LIN {X 0,Y 275.773,Z 716.506,A -85,B 0,C 180,E1 16932.937,E2 16932.937} C_VEL
LIN {X 0,Y 278.807,Z 722.231,A -85,B 0,C 180,E1 16937.514,E2 16937.514} C_VEL
LIN {X 0,Y 285.575,Z 736.206,A -85,B 0,C 180,E1 16944.998,E2 16944.998} C_VEL
LIN {X 0,Y 292.678,Z 753.38,A -85,B 0,C 180,E1 16951.647,E2 16951.647} C_VEL
LIN {X 0,Y 298.576,Z 772.807,A -85,B 0,C 180,E1 16957.666,E2 16957.666} C_VEL
LIN {X 0,Y 301.91,Z 794.325,A -85,B 0,C 180,E1 16963.416,E2 16963.416} C_VEL
LIN {X 0,Y 302.06,Z 807.18,A -85,B 0,C 180,E1 16966.628,E2 16966.628} C_VEL
LIN {X 0,Y 289.061,Z 835.016,A -85,B 0,C 180,E1 16971.838,E2 16971.838} C_VEL
LIN {X 0,Y 277.029,Z 857.298,A -85,B 0,C 180,E1 16977.972,E2 16977.972} C_VEL
LIN {X 0,Y 266.798,Z 875.138,A -85,B 0,C 180,E1 16985.37,E2 16985.37} C_VEL
LIN {X 0,Y 260.131,Z 886.98,A -85,B 0,C 180,E1 16993.139,E2 16993.139} C_VEL
LIN {X 0,Y 257.066,Z 893.034,A -85,B 0,C 180,E1 16999.857,E2 16999.857} C_VEL
LIN {X 0,Y 255.939,Z 895.924,A -85,B 0,C 180,E1 17006.62,E2 17006.62} C_VEL
LIN {X 0,Y 255.938,Z 895.892,A -85,B 0,C 180,E1 17013.38,E2 17013.38} C_VEL
LIN {X 0,Y 257.68,Z 891.722,A -85,B 0,C 180,E1 17021.827,E2 17021.827} C_VEL
LIN {X 0,Y 262.63,Z 882.447,A -85,B 0,C 180,E1 17030.166,E2 17030.166} C_VEL
LIN {X 0,Y 271.349,Z 867.242,A -85,B 0,C 180,E1 17038.209,E2 17038.209} C_VEL
LIN {X 0,Y 282.59,Z 847.082,A -85,B 0,C 180,E1 17045.032,E2 17045.032} C_VEL
LIN {X 0,Y 294.293,Z 824.104,A -85,B 0,C 180,E1 17050.34,E2 17050.34} C_VEL
LIN {X 0,Y 302.608,Z 805.568,A -85,B 0,C 180,E1 17053.512,E2 17053.512} C_VEL
LIN {X 0,Y 300.613,Z 783.565,A -85,B 0,C 180,E1 17059.276,E2 17059.276} C_VEL
LIN {X 0,Y 295.972,Z 763.231,A -85,B 0,C 180,E1 17065.01,E2 17065.01} C_VEL
LIN {X 0,Y 289.142,Z 744.349,A -85,B 0,C 180,E1 17071.442,E2 17071.442} C_VEL
LIN {X 0,Y 281.784,Z 728.351,A -85,B 0,C 180,E1 17078.651,E2 17078.651} C_VEL
LIN {X 0,Y 278.046,Z 721.516,A -85,B 0,C 180,E1 17083.047,E2 17083.047} C_VEL
LIN {X 0,Y 275.21,Z 715.444,A -85,B 0,C 180,E1 17087.74,E2 17087.74} C_VEL
LIN {X 0,Y 272.952,Z 711.906,A -85,B 0,C 180,E1 17098.422,E2 17098.422} C_VEL
LIN {X 0,Y 276.968,Z 716.793,A -85,B 0,C 180,E1 17107.559,E2 17107.559} C_VEL
LIN {X 0,Y 281.856,Z 725.008,A -85,B 0,C 180,E1 17113.023,E2 17113.023} C_VEL
LIN {X 0,Y 289.079,Z 736.426,A -85,B 0,C 180,E1 17118.645,E2 17118.645} C_VEL
LIN {X 0,Y 298.908,Z 754.882,A -85,B 0,C 180,E1 17124.806,E2 17124.806} C_VEL
LIN {X 0,Y 308.931,Z 777.729,A -85,B 0,C 180,E1 17130.453,E2 17130.453} C_VEL
LIN {X 0,Y 316.347,Z 802.298,A -85,B 0,C 180,E1 17135.213,E2 17135.213} C_VEL
LIN {X 0,Y 304.344,Z 840.414,A -85,B 0,C 180,E1 17138.476,E2 17138.476} C_VEL
LIN {X 0,Y 290.625,Z 875.361,A -85,B 0,C 180,E1 17142.899,E2 17142.899} C_VEL
LIN {X 0,Y 278.063,Z 904.903,A -85,B 0,C 180,E1 17148.334,E2 17148.334} C_VEL
LIN {X 0,Y 267.214,Z 930.489,A -85,B 0,C 180,E1 17154.988,E2 17154.988} C_VEL
LIN {X 0,Y 259.237,Z 951.979,A -85,B 0,C 180,E1 17162.904,E2 17162.904} C_VEL
LIN {X 0,Y 255.098,Z 967.514,A -85,B 0,C 180,E1 17171.173,E2 17171.173} C_VEL
LIN {X 0,Y 254.243,Z 975.961,A -85,B 0,C 180,E1 17177.835,E2 17177.835} C_VEL
LIN {X 0,Y 254.275,Z 980.166,A -85,B 0,C 180,E1 17183.183,E2 17183.183} C_VEL
LIN {X 0,Y 254.787,Z 982.267,A -85,B 0,C 180,E1 17190,E2 17190} C_VEL
LIN {X 0,Y 254.269,Z 980.175,A -85,B 0,C 180,E1 17196.817,E2 17196.817} C_VEL
LIN {X 0,Y 254.36,Z 973.333,A -85,B 0,C 180,E1 17204.604,E2 17204.604} C_VEL
LIN {X 0,Y 256.876,Z 959.841,A -85,B 0,C 180,E1 17213.361,E2 17213.361} C_VEL
LIN {X 0,Y 263.615,Z 939.724,A -85,B 0,C 180,E1 17221.971,E2 17221.971} C_VEL
LIN {X 0,Y 273.628,Z 915.458,A -85,B 0,C 180,E1 17229.203,E2 17229.203} C_VEL
LIN {X 0,Y 285.643,Z 887.471,A -85,B 0,C 180,E1 17235.11,E2 17235.11} C_VEL
LIN {X 0,Y 298.673,Z 855.592,A -85,B 0,C 180,E1 17239.823,E2 17239.823} C_VEL
LIN {X 0,Y 311.279,Z 820.186,A -85,B 0,C 180,E1 17243.408,E2 17243.408} C_VEL
LIN {X 0,Y 316.34,Z 802.002,A -85,B 0,C 180,E1 17244.859,E2 17244.859} C_VEL
LIN {X 0,Y 308.472,Z 776.099,A -85,B 0,C 180,E1 17249.903,E2 17249.903} C_VEL
LIN {X 0,Y 298.548,Z 753.828,A -85,B 0,C 180,E1 17255.505,E2 17255.505} C_VEL
LIN {X 0,Y 289.965,Z 738.122,A -85,B 0,C 180,E1 17260.822,E2 17260.822} C_VEL
LIN {X 0,Y 286.089,Z 736.306,A -85,B 0,C 180,E1 17262.977,E2 17262.977} C_VEL
LIN {X 0,Y 282.076,Z 736.045,A -85,B 0,C 180,E1 17265.282,E2 17265.282} C_VEL
LIN {X 0,Y 277.56,Z 729.06,A -85,B 0,C 180,E1 17269.674,E2 17269.674} C_VEL
LIN {X 0,Y 274.527,Z 723.198,A -85,B 0,C 180,E1 17274.079,E2 17274.079} C_VEL
LIN {X 0,Y 271.676,Z 719.971,A -85,B 0,C 180,E1 17281.181,E2 17281.181} C_VEL
LIN {X 0,Y 273.643,Z 723.735,A -85,B 0,C 180,E1 17292.432,E2 17292.432} C_VEL
LIN {X 0,Y 276.931,Z 731.578,A -85,B 0,C 180,E1 17298.252,E2 17298.252} C_VEL
LIN {X 0,Y 282.749,Z 744.678,A -85,B 0,C 180,E1 17305.266,E2 17305.266} C_VEL
LIN {X 0,Y 289.066,Z 761.562,A -85,B 0,C 180,E1 17311.901,E2 17311.901} C_VEL
LIN {X 0,Y 293.94,Z 781.055,A -85,B 0,C 180,E1 17318.017,E2 17318.017} C_VEL
LIN {X 0,Y 296.249,Z 803.118,A -85,B 0,C 180,E1 17324.083,E2 17324.083} C_VEL
LIN {X 0,Y 296.074,Z 809.506,A -85,B 0,C 180,E1 17325.739,E2 17325.739} C_VEL
LIN {X 0,Y 282.768,Z 836.72,A -85,B 0,C 180,E1 17330.943,E2 17330.943} C_VEL
LIN {X 0,Y 270.767,Z 858.109,A -85,B 0,C 180,E1 17336.916,E2 17336.916} C_VEL
LIN {X 0,Y 260.508,Z 875.122,A -85,B 0,C 180,E1 17343.949,E2 17343.949} C_VEL
LIN {X 0,Y 253.25,Z 887.277,A -85,B 0,C 180,E1 17351.771,E2 17351.771} C_VEL
LIN {X 0,Y 249.383,Z 894.348,A -85,B 0,C 180,E1 17359.541,E2 17359.541} C_VEL
LIN {X 0,Y 248.179,Z 897.233,A -85,B 0,C 180,E1 17366.514,E2 17366.514} C_VEL
LIN {X 0,Y 248.178,Z 897.201,A -85,B 0,C 180,E1 17373.486,E2 17373.486} C_VEL
LIN {X 0,Y 250.034,Z 893.041,A -85,B 0,C 180,E1 17382.194,E2 17382.194} C_VEL
LIN {X 0,Y 255.287,Z 883.772,A -85,B 0,C 180,E1 17390.772,E2 17390.772} C_VEL
LIN {X 0,Y 264.48,Z 868.573,A -85,B 0,C 180,E1 17399.01,E2 17399.01} C_VEL
LIN {X 0,Y 276.236,Z 848.436,A -85,B 0,C 180,E1 17405.961,E2 17405.961} C_VEL
LIN {X 0,Y 289.303,Z 823.666,A -85,B 0,C 180,E1 17411.685,E2 17411.685} C_VEL
LIN {X 0,Y 296.309,Z 807.713,A -85,B 0,C 180,E1 17414.535,E2 17414.535} C_VEL
LIN {X 0,Y 294.553,Z 785.102,A -85,B 0,C 180,E1 17420.725,E2 17420.725} C_VEL
LIN {X 0,Y 289.975,Z 764.717,A -85,B 0,C 180,E1 17426.887,E2 17426.887} C_VEL
LIN {X 0,Y 283.421,Z 746.135,A -85,B 0,C 180,E1 17433.851,E2 17433.851} C_VEL
LIN {X 0,Y 278.14,Z 734.597,A -85,B 0,C 180,E1 17439.737,E2 17439.737} C_VEL
LIN {X 0,Y 275.601,Z 728.908,A -85,B 0,C 180,E1 17443.302,E2 17443.302} C_VEL
LIN {X 0,Y 273.167,Z 723.013,A -85,B 0,C 180,E1 17448.052,E2 17448.052} C_VEL
LIN {X 0,Y 271.215,Z 719.663,A -85,B 0,C 180,E1 17456.817,E2 17456.817} C_VEL
LIN {X 0,Y 272.921,Z 722.001,A -85,B 0,C 180,E1 17463.622,E2 17463.622} C_VEL
LIN {X 0,Y 275.18,Z 724.57,A -85,B 0,C 180,E1 17467.311,E2 17467.311} C_VEL
LIN {X 0,Y 279.588,Z 732.408,A -85,B 0,C 180,E1 17472.652,E2 17472.652} C_VEL
LIN {X 0,Y 286.344,Z 743.669,A -85,B 0,C 180,E1 17478.239,E2 17478.239} C_VEL
LIN {X 0,Y 295.044,Z 760.875,A -85,B 0,C 180,E1 17484.156,E2 17484.156} C_VEL
LIN {X 0,Y 304.381,Z 783.881,A -85,B 0,C 180,E1 17490.025,E2 17490.025} C_VEL
LIN {X 0,Y 310.331,Z 804.847,A -85,B 0,C 180,E1 17494.246,E2 17494.246} C_VEL
LIN {X 0,Y 298.164,Z 841.829,A -85,B 0,C 180,E1 17497.569,E2 17497.569} C_VEL
LIN {X 0,Y 284.226,Z 875.806,A -85,B 0,C 180,E1 17501.989,E2 17501.989} C_VEL
LIN {X 0,Y 271.005,Z 905.4,A -85,B 0,C 180,E1 17507.607,E2 17507.607} C_VEL
LIN {X 0,Y 259.166,Z 932.085,A -85,B 0,C 180,E1 17514.902,E2 17514.902} C_VEL
LIN {X 0,Y 251.03,Z 953.123,A -85,B 0,C 180,E1 17523.202,E2 17523.202} C_VEL
LIN {X 0,Y 246.974,Z 968.527,A -85,B 0,C 180,E1 17532.212,E2 17532.212} C_VEL
LIN {X 0,Y 246.378,Z 976.356,A -85,B 0,C 180,E1 17539.412,E2 17539.412} C_VEL
LIN {X 0,Y 246.673,Z 980.374,A -85,B 0,C 180,E1 17546.493,E2 17546.493} C_VEL
LIN {X 0,Y 246.995,Z 980.955,A -85,B 0,C 180,E1 17550,E2 17550} C_VEL
LIN {X 0,Y 246.432,Z 978.846,A -85,B 0,C 180,E1 17557.035,E2 17557.035} C_VEL
LIN {X 0,Y 246.568,Z 971.973,A -85,B 0,C 180,E1 17565.076,E2 17565.076} C_VEL
LIN {X 0,Y 249.374,Z 958.451,A -85,B 0,C 180,E1 17574.107,E2 17574.107} C_VEL
LIN {X 0,Y 256.602,Z 938.302,A -85,B 0,C 180,E1 17582.954,E2 17582.954} C_VEL
LIN {X 0,Y 266.993,Z 914.605,A -85,B 0,C 180,E1 17590.179,E2 17590.179} C_VEL
LIN {X 0,Y 280.023,Z 885.552,A -85,B 0,C 180,E1 17596.396,E2 17596.396} C_VEL
LIN {X 0,Y 293.699,Z 853.458,A -85,B 0,C 180,E1 17601.123,E2 17601.123} C_VEL
LIN {X 0,Y 307.066,Z 816.863,A -85,B 0,C 180,E1 17604.776,E2 17604.776} C_VEL
LIN {X 0,Y 310.458,Z 805.145,A -85,B 0,C 180,E1 17605.719,E2 17605.719} C_VEL
LIN {X 0,Y 303.059,Z 779.517,A -85,B 0,C 180,E1 17610.953,E2 17610.953} C_VEL
LIN {X 0,Y 293.585,Z 757.473,A -85,B 0,C 180,E1 17616.879,E2 17616.879} C_VEL
LIN {X 0,Y 284.72,Z 740.905,A -85,B 0,C 180,E1 17623.072,E2 17623.072} C_VEL
LIN {X 0,Y 282.076,Z 736.045,A -85,B 0,C 180,E1 17625.282,E2 17625.282} C_VEL
LIN {X 0,Y 273.842,Z 734.194,A -85,B 0,C 180,E1 17631.882,E2 17631.882} C_VEL
LIN {X 0,Y 273.556,Z 733.6,A -85,B 0,C 180,E1 17632.32,E2 17632.32} C_VEL
LIN {X 0,Y 272.416,Z 730.73,A -85,B 0,C 180,E1 17634.431,E2 17634.431} C_VEL
LIN {X 0,Y 269.829,Z 727.655,A -85,B 0,C 180,E1 17641.189,E2 17641.189} C_VEL
LIN {X 0,Y 271.298,Z 731.406,A -85,B 0,C 180,E1 17652.236,E2 17652.236} C_VEL
LIN {X 0,Y 276.241,Z 743.627,A -85,B 0,C 180,E1 17660.957,E2 17660.957} C_VEL
LIN {X 0,Y 282.102,Z 759.424,A -85,B 0,C 180,E1 17668.333,E2 17668.333} C_VEL
LIN {X 0,Y 287.086,Z 777.8,A -85,B 0,C 180,E1 17674.862,E2 17674.862} C_VEL
LIN {X 0,Y 289.601,Z 795.656,A -85,B 0,C 180,E1 17680.221,E2 17680.221} C_VEL
LIN {X 0,Y 289.774,Z 812.608,A -85,B 0,C 180,E1 17684.944,E2 17684.944} C_VEL
LIN {X 0,Y 276.676,Z 838.218,A -85,B 0,C 180,E1 17689.961,E2 17689.961} C_VEL
LIN {X 0,Y 264.236,Z 859.448,A -85,B 0,C 180,E1 17695.988,E2 17695.988} C_VEL
LIN {X 0,Y 252.723,Z 877.646,A -85,B 0,C 180,E1 17703.809,E2 17703.809} C_VEL
LIN {X 0,Y 245.203,Z 889.619,A -85,B 0,C 180,E1 17712.079,E2 17712.079} C_VEL
LIN {X 0,Y 241.706,Z 895.663,A -85,B 0,C 180,E1 17719.205,E2 17719.205} C_VEL
LIN {X 0,Y 240.404,Z 898.544,A -85,B 0,C 180,E1 17726.401,E2 17726.401} C_VEL
LIN {X 0,Y 240.404,Z 898.513,A -85,B 0,C 180,E1 17733.599,E2 17733.599} C_VEL
LIN {X 0,Y 242.405,Z 894.357,A -85,B 0,C 180,E1 17742.584,E2 17742.584} C_VEL
LIN {X 0,Y 247.994,Z 885.093,A -85,B 0,C 180,E1 17751.413,E2 17751.413} C_VEL
LIN {X 0,Y 257.672,Z 869.902,A -85,B 0,C 180,E1 17759.853,E2 17759.853} C_VEL
LIN {X 0,Y 269.956,Z 849.787,A -85,B 0,C 180,E1 17766.934,E2 17766.934} C_VEL
LIN {X 0,Y 283.533,Z 825.049,A -85,B 0,C 180,E1 17772.732,E2 17772.732} C_VEL
LIN {X 0,Y 290.1,Z 810.596,A -85,B 0,C 180,E1 17775.402,E2 17775.402} C_VEL
LIN {X 0,Y 288.869,Z 788.876,A -85,B 0,C 180,E1 17781.589,E2 17781.589} C_VEL
LIN {X 0,Y 285.281,Z 770.474,A -85,B 0,C 180,E1 17787.424,E2 17787.424} C_VEL
LIN {X 0,Y 279.61,Z 752.493,A -85,B 0,C 180,E1 17794.43,E2 17794.43} C_VEL
LIN {X 0,Y 274.685,Z 740.648,A -85,B 0,C 180,E1 17800.763,E2 17800.763} C_VEL
LIN {X 0,Y 272.75,Z 735.962,A -85,B 0,C 180,E1 17803.949,E2 17803.949} C_VEL
LIN {X 0,Y 270.656,Z 730.403,A -85,B 0,C 180,E1 17808.754,E2 17808.754} C_VEL
LIN {X 0,Y 269.534,Z 727.451,A -85,B 0,C 180,E1 17818.402,E2 17818.402} C_VEL
LIN {X 0,Y 272.989,Z 731.942,A -85,B 0,C 180,E1 17826.891,E2 17826.891} C_VEL
LIN {X 0,Y 277.382,Z 740.093,A -85,B 0,C 180,E1 17832.474,E2 17832.474} C_VEL
LIN {X 0,Y 283.65,Z 751.509,A -85,B 0,C 180,E1 17838.117,E2 17838.117} C_VEL
LIN {X 0,Y 292.288,Z 769.765,A -85,B 0,C 180,E1 17844.399,E2 17844.399} C_VEL
LIN {X 0,Y 299.943,Z 790.603,A -85,B 0,C 180,E1 17849.727,E2 17849.727} C_VEL
LIN {X 0,Y 304.516,Z 808.446,A -85,B 0,C 180,E1 17853.46,E2 17853.46} C_VEL
LIN {X 0,Y 291.73,Z 844.092,A -85,B 0,C 180,E1 17856.717,E2 17856.717} C_VEL
LIN {X 0,Y 277.252,Z 877.65,A -85,B 0,C 180,E1 17861.256,E2 17861.256} C_VEL
LIN {X 0,Y 262.431,Z 909.204,A -85,B 0,C 180,E1 17867.636,E2 17867.636} C_VEL
LIN {X 0,Y 250.611,Z 934.587,A -85,B 0,C 180,E1 17875.189,E2 17875.189} C_VEL
LIN {X 0,Y 242.975,Z 953.491,A -85,B 0,C 180,E1 17883.24,E2 17883.24} C_VEL
LIN {X 0,Y 239.025,Z 968.3,A -85,B 0,C 180,E1 17892.55,E2 17892.55} C_VEL
LIN {X 0,Y 238.545,Z 976.432,A -85,B 0,C 180,E1 17900.901,E2 17900.901} C_VEL
LIN {X 0,Y 238.866,Z 979.056,A -85,B 0,C 180,E1 17906.378,E2 17906.378} C_VEL
LIN {X 0,Y 239.194,Z 979.642,A -85,B 0,C 180,E1 17910,E2 17910} C_VEL
LIN {X 0,Y 238.593,Z 977.515,A -85,B 0,C 180,E1 17917.267,E2 17917.267} C_VEL
LIN {X 0,Y 238.805,Z 970.615,A -85,B 0,C 180,E1 17925.578,E2 17925.578} C_VEL
LIN {X 0,Y 241.829,Z 957.133,A -85,B 0,C 180,E1 17934.862,E2 17934.862} C_VEL
LIN {X 0,Y 249.599,Z 936.935,A -85,B 0,C 180,E1 17943.976,E2 17943.976} C_VEL
LIN {X 0,Y 260.742,Z 913.024,A -85,B 0,C 180,E1 17951.395,E2 17951.395} C_VEL
LIN {X 0,Y 273.892,Z 885.103,A -85,B 0,C 180,E1 17957.467,E2 17957.467} C_VEL
LIN {X 0,Y 288.069,Z 853.225,A -85,B 0,C 180,E1 17962.234,E2 17962.234} C_VEL
LIN {X 0,Y 301.44,Z 818.115,A -85,B 0,C 180,E1 17965.798,E2 17965.798} C_VEL
LIN {X 0,Y 304.447,Z 807.665,A -85,B 0,C 180,E1 17966.71,E2 17966.71} C_VEL
LIN {X 0,Y 297.663,Z 783.084,A -85,B 0,C 180,E1 17972.031,E2 17972.031} C_VEL
LIN {X 0,Y 289.298,Z 762.856,A -85,B 0,C 180,E1 17977.776,E2 17977.776} C_VEL
LIN {X 0,Y 281.617,Z 747.621,A -85,B 0,C 180,E1 17983.669,E2 17983.669} C_VEL
LIN {X 0,Y 275.493,Z 736.621,A -85,B 0,C 180,E1 17989.831,E2 17989.831} C_VEL
LIN {X 0,Y 273.556,Z 733.6,A -85,B 0,C 180,E1 17992.32,E2 17992.32} C_VEL
LIN {X 0,Y 271.902,Z 733.916,A -85,B 0,C 180,E1 17994.118,E2 17994.118} C_VEL
LIN {X 0,Y 269.049,Z 737.187,A -85,B 0,C 180,E1 17996.855,E2 17996.855} C_VEL
LIN {X 0,Y 268.887,Z 737.1,A -85,B 0,C 180,E1 17997.174,E2 17997.174} C_VEL
LIN {X 0,Y 267.483,Z 735.272,A -85,B 0,C 180,E1 18003.228,E2 18003.228} C_VEL
LIN {X 0,Y 268.824,Z 739.224,A -85,B 0,C 180,E1 18012.144,E2 18012.144} C_VEL
LIN {X 0,Y 272.607,Z 749.793,A -85,B 0,C 180,E1 18020.096,E2 18020.096} C_VEL
LIN {X 0,Y 277.39,Z 764.046,A -85,B 0,C 180,E1 18027.168,E2 18027.168} C_VEL
LIN {X 0,Y 281.67,Z 781.506,A -85,B 0,C 180,E1 18033.757,E2 18033.757} C_VEL
LIN {X 0,Y 283.808,Z 800.155,A -85,B 0,C 180,E1 18039.634,E2 18039.634} C_VEL
LIN {X 0,Y 283.745,Z 815.144,A -85,B 0,C 180,E1 18044.028,E2 18044.028} C_VEL
LIN {X 0,Y 270.039,Z 840.765,A -85,B 0,C 180,E1 18049.189,E2 18049.189} C_VEL
LIN {X 0,Y 256.886,Z 862.177,A -85,B 0,C 180,E1 18055.518,E2 18055.518} C_VEL
LIN {X 0,Y 245.244,Z 879.716,A -85,B 0,C 180,E1 18063.413,E2 18063.413} C_VEL
LIN {X 0,Y 236.918,Z 892.249,A -85,B 0,C 180,E1 18072.784,E2 18072.784} C_VEL
LIN {X 0,Y 233.073,Z 898.782,A -85,B 0,C 180,E1 18082.56,E2 18082.56} C_VEL
LIN {X 0,Y 232.297,Z 900.265,A -85,B 0,C 180,E1 18090,E2 18090} C_VEL
LIN {X 0,Y 233.075,Z 898.729,A -85,B 0,C 180,E1 18097.44,E2 18097.44} C_VEL
LIN {X 0,Y 237.02,Z 892.057,A -85,B 0,C 180,E1 18107.295,E2 18107.295} C_VEL
LIN {X 0,Y 245.408,Z 879.388,A -85,B 0,C 180,E1 18116.639,E2 18116.639} C_VEL
LIN {X 0,Y 257.207,Z 861.555,A -85,B 0,C 180,E1 18124.586,E2 18124.586} C_VEL
LIN {X 0,Y 270.968,Z 838.952,A -85,B 0,C 180,E1 18131.15,E2 18131.15} C_VEL
LIN {X 0,Y 283.915,Z 814.155,A -85,B 0,C 180,E1 18136.091,E2 18136.091} C_VEL
LIN {X 0,Y 283.262,Z 792.822,A -85,B 0,C 180,E1 18142.432,E2 18142.432} C_VEL
LIN {X 0,Y 279.983,Z 773.942,A -85,B 0,C 180,E1 18148.762,E2 18148.762} C_VEL
LIN {X 0,Y 275.729,Z 758.969,A -85,B 0,C 180,E1 18154.913,E2 18154.913} C_VEL
LIN {X 0,Y 270.832,Z 744.586,A -85,B 0,C 180,E1 18162.916,E2 18162.916} C_VEL
LIN {X 0,Y 268.459,Z 737.983,A -85,B 0,C 180,E1 18168.661,E2 18168.661} C_VEL
LIN {X 0,Y 267.498,Z 735.067,A -85,B 0,C 180,E1 18178.39,E2 18178.39} C_VEL
LIN {X 0,Y 270.718,Z 739.485,A -85,B 0,C 180,E1 18186.607,E2 18186.607} C_VEL
LIN {X 0,Y 274.933,Z 747.802,A -85,B 0,C 180,E1 18192.385,E2 18192.385} C_VEL
LIN {X 0,Y 281.753,Z 760.881,A -85,B 0,C 180,E1 18198.749,E2 18198.749} C_VEL
LIN {X 0,Y 289.78,Z 780.082,A -85,B 0,C 180,E1 18205.077,E2 18205.077} C_VEL
LIN {X 0,Y 296.653,Z 802.266,A -85,B 0,C 180,E1 18210.579,E2 18210.579} C_VEL
LIN {X 0,Y 298.485,Z 811.961,A -85,B 0,C 180,E1 18212.564,E2 18212.564} C_VEL
LIN {X 0,Y 284.132,Z 849.211,A -85,B 0,C 180,E1 18216.165,E2 18216.165} C_VEL
LIN {X 0,Y 268.819,Z 882.478,A -85,B 0,C 180,E1 18221.036,E2 18221.036} C_VEL
LIN {X 0,Y 254.307,Z 911.835,A -85,B 0,C 180,E1 18227.444,E2 18227.444} C_VEL
LIN {X 0,Y 242.454,Z 936.101,A -85,B 0,C 180,E1 18235.17,E2 18235.17} C_VEL
LIN {X 0,Y 234.193,Z 955.97,A -85,B 0,C 180,E1 18244.439,E2 18244.439} C_VEL
LIN {X 0,Y 230.969,Z 969.219,A -85,B 0,C 180,E1 18253.879,E2 18253.879} C_VEL
LIN {X 0,Y 230.764,Z 976.174,A -85,B 0,C 180,E1 18262.485,E2 18262.485} C_VEL
LIN {X 0,Y 231.4,Z 978.33,A -85,B 0,C 180,E1 18270,E2 18270} C_VEL
LIN {X 0,Y 230.754,Z 976.184,A -85,B 0,C 180,E1 18277.515,E2 18277.515} C_VEL
LIN {X 0,Y 231.002,Z 969.247,A -85,B 0,C 180,E1 18286.119,E2 18286.119} C_VEL
LIN {X 0,Y 234.545,Z 955.112,A -85,B 0,C 180,E1 18296.05,E2 18296.05} C_VEL
LIN {X 0,Y 242.414,Z 936.109,A -85,B 0,C 180,E1 18304.854,E2 18304.854} C_VEL
LIN {X 0,Y 254.876,Z 910.809,A -85,B 0,C 180,E1 18312.845,E2 18312.845} C_VEL
LIN {X 0,Y 268.914,Z 882.626,A -85,B 0,C 180,E1 18318.941,E2 18318.941} C_VEL
LIN {X 0,Y 283.532,Z 850.753,A -85,B 0,C 180,E1 18323.667,E2 18323.667} C_VEL
LIN {X 0,Y 297.869,Z 814.005,A -85,B 0,C 180,E1 18327.3,E2 18327.3} C_VEL
LIN {X 0,Y 298.219,Z 808.718,A -85,B 0,C 180,E1 18328.043,E2 18328.043} C_VEL
LIN {X 0,Y 291.884,Z 785.192,A -85,B 0,C 180,E1 18333.519,E2 18333.519} C_VEL
LIN {X 0,Y 283.675,Z 765.047,A -85,B 0,C 180,E1 18339.767,E2 18339.767} C_VEL
LIN {X 0,Y 276.216,Z 749.889,A -85,B 0,C 180,E1 18346.469,E2 18346.469} C_VEL
LIN {X 0,Y 272.499,Z 743.381,A -85,B 0,C 180,E1 18350.733,E2 18350.733} C_VEL
LIN {X 0,Y 270.161,Z 738.234,A -85,B 0,C 180,E1 18354.787,E2 18354.787} C_VEL
LIN {X 0,Y 268.887,Z 737.1,A -85,B 0,C 180,E1 18357.174,E2 18357.174} C_VEL
LIN {X 0,Y 267.305,Z 738.248,A -85,B 0,C 180,E1 18359.937,E2 18359.937} C_VEL
LIN {X 0,Y 265.042,Z 743.301,A -85,B 0,C 180,E1 18364.565,E2 18364.565} C_VEL
LIN {X 0,Y 266.082,Z 745.892,A -85,B 0,C 180,E1 18371.335,E2 18371.335} C_VEL
LIN {X 0,Y 269.217,Z 756.616,A -85,B 0,C 180,E1 18379.644,E2 18379.644} C_VEL
LIN {X 0,Y 273.203,Z 770.441,A -85,B 0,C 180,E1 18386.745,E2 18386.745} C_VEL
LIN {X 0,Y 276.695,Z 787.513,A -85,B 0,C 180,E1 18393.415,E2 18393.415} C_VEL
LIN {X 0,Y 278.058,Z 804.942,A -85,B 0,C 180,E1 18399.113,E2 18399.113} C_VEL
LIN {X 0,Y 277.595,Z 818.011,A -85,B 0,C 180,E1 18403.121,E2 18403.121} C_VEL
LIN {X 0,Y 263.019,Z 844.041,A -85,B 0,C 180,E1 18408.562,E2 18408.562} C_VEL
LIN {X 0,Y 248.596,Z 866.341,A -85,B 0,C 180,E1 18415.552,E2 18415.552} C_VEL
LIN {X 0,Y 237.16,Z 882.652,A -85,B 0,C 180,E1 18423.552,E2 18423.552} C_VEL
LIN {X 0,Y 229.46,Z 893.567,A -85,B 0,C 180,E1 18432.206,E2 18432.206} C_VEL
LIN {X 0,Y 225.329,Z 900.097,A -85,B 0,C 180,E1 18442.303,E2 18442.303} C_VEL
LIN {X 0,Y 224.537,Z 901.572,A -85,B 0,C 180,E1 18450,E2 18450} C_VEL
LIN {X 0,Y 225.333,Z 900.045,A -85,B 0,C 180,E1 18457.697,E2 18457.697} C_VEL
LIN {X 0,Y 229.569,Z 893.374,A -85,B 0,C 180,E1 18467.875,E2 18467.875} C_VEL
LIN {X 0,Y 238.192,Z 881.066,A -85,B 0,C 180,E1 18477.289,E2 18477.289} C_VEL
LIN {X 0,Y 249.824,Z 864.392,A -85,B 0,C 180,E1 18485.045,E2 18485.045} C_VEL
LIN {X 0,Y 263.223,Z 843.437,A -85,B 0,C 180,E1 18491.488,E2 18491.488} C_VEL
LIN {X 0,Y 277.695,Z 817.608,A -85,B 0,C 180,E1 18496.831,E2 18496.831} C_VEL
LIN {X 0,Y 277.819,Z 798.36,A -85,B 0,C 180,E1 18502.813,E2 18502.813} C_VEL
LIN {X 0,Y 275.261,Z 779.684,A -85,B 0,C 180,E1 18509.314,E2 18509.314} C_VEL
LIN {X 0,Y 271.483,Z 764.455,A -85,B 0,C 180,E1 18515.896,E2 18515.896} C_VEL
LIN {X 0,Y 267.509,Z 751.28,A -85,B 0,C 180,E1 18523.625,E2 18523.625} C_VEL
LIN {X 0,Y 265.849,Z 745.557,A -85,B 0,C 180,E1 18528.743,E2 18528.743} C_VEL
LIN {X 0,Y 265.074,Z 742.573,A -85,B 0,C 180,E1 18536.743,E2 18536.743} C_VEL
LIN {X 0,Y 266.857,Z 744.948,A -85,B 0,C 180,E1 18543.653,E2 18543.653} C_VEL
LIN {X 0,Y 268.383,Z 747.304,A -85,B 0,C 180,E1 18546.564,E2 18546.564} C_VEL
LIN {X 0,Y 272.079,Z 754.944,A -85,B 0,C 180,E1 18552.009,E2 18552.009} C_VEL
LIN {X 0,Y 278.188,Z 767.353,A -85,B 0,C 180,E1 18558.179,E2 18558.179} C_VEL
LIN {X 0,Y 285.57,Z 786.589,A -85,B 0,C 180,E1 18564.682,E2 18564.682} C_VEL
LIN {X 0,Y 291.327,Z 807.134,A -85,B 0,C 180,E1 18569.953,E2 18569.953} C_VEL
LIN {X 0,Y 292.446,Z 815.103,A -85,B 0,C 180,E1 18571.603,E2 18571.603} C_VEL
LIN {X 0,Y 278.536,Z 849.498,A -85,B 0,C 180,E1 18575.025,E2 18575.025} C_VEL
LIN {X 0,Y 263.479,Z 880.999,A -85,B 0,C 180,E1 18579.679,E2 18579.679} C_VEL
LIN {X 0,Y 248.046,Z 910.675,A -85,B 0,C 180,E1 18586.214,E2 18586.214} C_VEL
LIN {X 0,Y 235.573,Z 934.794,A -85,B 0,C 180,E1 18594.056,E2 18594.056} C_VEL
LIN {X 0,Y 226.593,Z 954.953,A -85,B 0,C 180,E1 18603.767,E2 18603.767} C_VEL
LIN {X 0,Y 223.296,Z 966.997,A -85,B 0,C 180,E1 18612.556,E2 18612.556} C_VEL
LIN {X 0,Y 222.911,Z 973.944,A -85,B 0,C 180,E1 18620.581,E2 18620.581} C_VEL
LIN {X 0,Y 223.223,Z 976.416,A -85,B 0,C 180,E1 18626.124,E2 18626.124} C_VEL
LIN {X 0,Y 223.627,Z 977.021,A -85,B 0,C 180,E1 18630,E2 18630} C_VEL
LIN {X 0,Y 222.918,Z 974.853,A -85,B 0,C 180,E1 18637.781,E2 18637.781} C_VEL
LIN {X 0,Y 223.099,Z 968.855,A -85,B 0,C 180,E1 18645.697,E2 18645.697} C_VEL
LIN {X 0,Y 226.36,Z 955.934,A -85,B 0,C 180,E1 18655.632,E2 18655.632} C_VEL
LIN {X 0,Y 234.789,Z 936.424,A -85,B 0,C 180,E1 18665.34,E2 18665.34} C_VEL
LIN {X 0,Y 247.77,Z 911.388,A -85,B 0,C 180,E1 18673.614,E2 18673.614} C_VEL
LIN {X 0,Y 262.707,Z 882.848,A -85,B 0,C 180,E1 18679.989,E2 18679.989} C_VEL
LIN {X 0,Y 278.004,Z 850.891,A -85,B 0,C 180,E1 18684.822,E2 18684.822} C_VEL
LIN {X 0,Y 292.545,Z 815.106,A -85,B 0,C 180,E1 18688.415,E2 18688.415} C_VEL
LIN {X 0,Y 288.89,Z 796.484,A -85,B 0,C 180,E1 18692.62,E2 18692.62} C_VEL
LIN {X 0,Y 282.096,Z 776.697,A -85,B 0,C 180,E1 18698.418,E2 18698.418} C_VEL
LIN {X 0,Y 275.855,Z 762.283,A -85,B 0,C 180,E1 18704.122,E2 18704.122} C_VEL
LIN {X 0,Y 270.475,Z 751.392,A -85,B 0,C 180,E1 18710.36,E2 18710.36} C_VEL
LIN {X 0,Y 267.717,Z 745.676,A -85,B 0,C 180,E1 18715.144,E2 18715.144} C_VEL
LIN {X 0,Y 265.247,Z 742.864,A -85,B 0,C 180,E1 18723.255,E2 18723.255} C_VEL
LIN {X 0,Y 265.042,Z 743.301,A -85,B 0,C 180,E1 18724.565,E2 18724.565} C_VEL
LIN {X 0,Y 264.041,Z 747.941,A -85,B 0,C 180,E1 18728.201,E2 18728.201} C_VEL
LIN {X 0,Y 263.255,Z 754.165,A -85,B 0,C 180,E1 18731.804,E2 18731.804} C_VEL
LIN {X 0,Y 265.925,Z 764.535,A -85,B 0,C 180,E1 18739.897,E2 18739.897} C_VEL
LIN {X 0,Y 269.28,Z 778.628,A -85,B 0,C 180,E1 18747.166,E2 18747.166} C_VEL
LIN {X 0,Y 271.755,Z 795.257,A -85,B 0,C 180,E1 18753.72,E2 18753.72} C_VEL
LIN {X 0,Y 272.131,Z 813.519,A -85,B 0,C 180,E1 18759.84,E2 18759.84} C_VEL
LIN {X 0,Y 271.666,Z 820.651,A -85,B 0,C 180,E1 18762.143,E2 18762.143} C_VEL
LIN {X 0,Y 256.935,Z 845.874,A -85,B 0,C 180,E1 18767.537,E2 18767.537} C_VEL
LIN {X 0,Y 242.186,Z 867.688,A -85,B 0,C 180,E1 18774.514,E2 18774.514} C_VEL
LIN {X 0,Y 230.149,Z 883.979,A -85,B 0,C 180,E1 18782.68,E2 18782.68} C_VEL
LIN {X 0,Y 221.4,Z 895.726,A -85,B 0,C 180,E1 18792.553,E2 18792.553} C_VEL
LIN {X 0,Y 217.607,Z 901.409,A -85,B 0,C 180,E1 18802.028,E2 18802.028} C_VEL
LIN {X 0,Y 216.754,Z 902.882,A -85,B 0,C 180,E1 18810,E2 18810} C_VEL
LIN {X 0,Y 217.613,Z 901.357,A -85,B 0,C 180,E1 18817.972,E2 18817.972} C_VEL
LIN {X 0,Y 222.005,Z 894.869,A -85,B 0,C 180,E1 18828.289,E2 18828.289} C_VEL
LIN {X 0,Y 231.117,Z 882.614,A -85,B 0,C 180,E1 18838.049,E2 18838.049} C_VEL
LIN {X 0,Y 243.532,Z 865.622,A -85,B 0,C 180,E1 18846.143,E2 18846.143} C_VEL
LIN {X 0,Y 257.767,Z 844.259,A -85,B 0,C 180,E1 18852.773,E2 18852.773} C_VEL
LIN {X 0,Y 271.637,Z 820.263,A -85,B 0,C 180,E1 18857.846,E2 18857.846} C_VEL
LIN {X 0,Y 272.169,Z 801.454,A -85,B 0,C 180,E1 18863.962,E2 18863.962} C_VEL
LIN {X 0,Y 270.149,Z 783.516,A -85,B 0,C 180,E1 18870.613,E2 18870.613} C_VEL
LIN {X 0,Y 266.94,Z 768.407,A -85,B 0,C 180,E1 18877.577,E2 18877.577} C_VEL
LIN {X 0,Y 264.165,Z 757.956,A -85,B 0,C 180,E1 18884.39,E2 18884.39} C_VEL
LIN {X 0,Y 262.733,Z 752.4,A -85,B 0,C 180,E1 18890.085,E2 18890.085} C_VEL
LIN {X 0,Y 262.536,Z 750.097,A -85,B 0,C 180,E1 18896.712,E2 18896.712} C_VEL
LIN {X 0,Y 264.183,Z 752.267,A -85,B 0,C 180,E1 18903.28,E2 18903.28} C_VEL
LIN {X 0,Y 265.727,Z 755.034,A -85,B 0,C 180,E1 18906.527,E2 18906.527} C_VEL
LIN {X 0,Y 270.166,Z 764.037,A -85,B 0,C 180,E1 18912.915,E2 18912.915} C_VEL
LIN {X 0,Y 276.726,Z 779.701,A -85,B 0,C 180,E1 18919.931,E2 18919.931} C_VEL
LIN {X 0,Y 283.252,Z 799.989,A -85,B 0,C 180,E1 18926.293,E2 18926.293} C_VEL
LIN {X 0,Y 286.771,Z 816.344,A -85,B 0,C 180,E1 18930.351,E2 18930.351} C_VEL
LIN {X 0,Y 272.177,Z 851.752,A -85,B 0,C 180,E1 18934.09,E2 18934.09} C_VEL
LIN {X 0,Y 256.223,Z 883.384,A -85,B 0,C 180,E1 18938.969,E2 18938.969} C_VEL
LIN {X 0,Y 240.392,Z 912.383,A -85,B 0,C 180,E1 18945.706,E2 18945.706} C_VEL
LIN {X 0,Y 226.948,Z 937.169,A -85,B 0,C 180,E1 18954.423,E2 18954.423} C_VEL
LIN {X 0,Y 218.582,Z 955.113,A -85,B 0,C 180,E1 18963.835,E2 18963.835} C_VEL
LIN {X 0,Y 215.259,Z 967.458,A -85,B 0,C 180,E1 18973.716,E2 18973.716} C_VEL
LIN {X 0,Y 215.097,Z 973.51,A -85,B 0,C 180,E1 18981.934,E2 18981.934} C_VEL
LIN {X 0,Y 215.83,Z 975.708,A -85,B 0,C 180,E1 18990,E2 18990} C_VEL
LIN {X 0,Y 215.087,Z 973.522,A -85,B 0,C 180,E1 18998.066,E2 18998.066} C_VEL
LIN {X 0,Y 215.296,Z 967.488,A -85,B 0,C 180,E1 19006.281,E2 19006.281} C_VEL
LIN {X 0,Y 218.722,Z 955.036,A -85,B 0,C 180,E1 19016.24,E2 19016.24} C_VEL
LIN {X 0,Y 227.435,Z 936.115,A -85,B 0,C 180,E1 19026.075,E2 19026.075} C_VEL
LIN {X 0,Y 241.252,Z 910.905,A -85,B 0,C 180,E1 19034.722,E2 19034.722} C_VEL
LIN {X 0,Y 257.203,Z 881.789,A -85,B 0,C 180,E1 19041.335,E2 19041.335} C_VEL
LIN {X 0,Y 273.301,Z 849.549,A -85,B 0,C 180,E1 19046.203,E2 19046.203} C_VEL
LIN {X 0,Y 286.878,Z 816.371,A -85,B 0,C 180,E1 19049.664,E2 19049.664} C_VEL
LIN {X 0,Y 282.143,Z 795.229,A -85,B 0,C 180,E1 19055.044,E2 19055.044} C_VEL
LIN {X 0,Y 276.034,Z 777.812,A -85,B 0,C 180,E1 19060.848,E2 19060.848} C_VEL
LIN {X 0,Y 270.331,Z 764.159,A -85,B 0,C 180,E1 19067.093,E2 19067.093} C_VEL
LIN {X 0,Y 265.249,Z 753.178,A -85,B 0,C 180,E1 19075.099,E2 19075.099} C_VEL
LIN {X 0,Y 262.718,Z 750.364,A -85,B 0,C 180,E1 19083.286,E2 19083.286} C_VEL
LIN {X 0,Y 263.255,Z 754.165,A -85,B 0,C 180,E1 19091.804,E2 19091.804} C_VEL
LIN {X 0,Y 262.474,Z 761.803,A -85,B 0,C 180,E1 19095.245,E2 19095.245} C_VEL
LIN {X 0,Y 261.913,Z 769.961,A -85,B 0,C 180,E1 19098.676,E2 19098.676} C_VEL
LIN {X 0,Y 264.462,Z 782.746,A -85,B 0,C 180,E1 19105.776,E2 19105.776} C_VEL
LIN {X 0,Y 266.367,Z 798.683,A -85,B 0,C 180,E1 19112.485,E2 19112.485} C_VEL
LIN {X 0,Y 266.349,Z 815.782,A -85,B 0,C 180,E1 19118.539,E2 19118.539} C_VEL
LIN {X 0,Y 265.152,Z 824.511,A -85,B 0,C 180,E1 19121.336,E2 19121.336} C_VEL
LIN {X 0,Y 248.726,Z 850.939,A -85,B 0,C 180,E1 19127.337,E2 19127.337} C_VEL
LIN {X 0,Y 233.866,Z 871.56,A -85,B 0,C 180,E1 19134.499,E2 19134.499} C_VEL
LIN {X 0,Y 221.072,Z 888.066,A -85,B 0,C 180,E1 19143.661,E2 19143.661} C_VEL
LIN {X 0,Y 213.036,Z 898.354,A -85,B 0,C 180,E1 19153.541,E2 19153.541} C_VEL
LIN {X 0,Y 209.872,Z 902.724,A -85,B 0,C 180,E1 19161.732,E2 19161.732} C_VEL
LIN {X 0,Y 208.965,Z 904.193,A -85,B 0,C 180,E1 19170,E2 19170} C_VEL
LIN {X 0,Y 209.904,Z 902.668,A -85,B 0,C 180,E1 19178.267,E2 19178.267} C_VEL
LIN {X 0,Y 214.852,Z 895.877,A -85,B 0,C 180,E1 19189.312,E2 19189.312} C_VEL
LIN {X 0,Y 224.263,Z 883.907,A -85,B 0,C 180,E1 19199.01,E2 19199.01} C_VEL
LIN {X 0,Y 237.266,Z 866.96,A -85,B 0,C 180,E1 19207.256,E2 19207.256} C_VEL
LIN {X 0,Y 251.712,Z 846.212,A -85,B 0,C 180,E1 19213.825,E2 19213.825} C_VEL
LIN {X 0,Y 265.635,Z 823.117,A -85,B 0,C 180,E1 19218.845,E2 19218.845} C_VEL
LIN {X 0,Y 266.551,Z 804.99,A -85,B 0,C 180,E1 19225.037,E2 19225.037} C_VEL
LIN {X 0,Y 265.205,Z 788.286,A -85,B 0,C 180,E1 19231.55,E2 19231.55} C_VEL
LIN {X 0,Y 262.844,Z 774.459,A -85,B 0,C 180,E1 19238.299,E2 19238.299} C_VEL
LIN {X 0,Y 260.712,Z 764.752,A -85,B 0,C 180,E1 19244.91,E2 19244.91} C_VEL
LIN {X 0,Y 259.633,Z 759.408,A -85,B 0,C 180,E1 19251.13,E2 19251.13} C_VEL
LIN {X 0,Y 259.824,Z 757.561,A -85,B 0,C 180,E1 19256.677,E2 19256.677} C_VEL
LIN {X 0,Y 261.572,Z 759.72,A -85,B 0,C 180,E1 19263.313,E2 19263.313} C_VEL
LIN {X 0,Y 262.982,Z 762.768,A -85,B 0,C 180,E1 19266.596,E2 19266.596} C_VEL
LIN {X 0,Y 267.184,Z 771.907,A -85,B 0,C 180,E1 19273.062,E2 19273.062} C_VEL
LIN {X 0,Y 272.877,Z 786.962,A -85,B 0,C 180,E1 19279.77,E2 19279.77} C_VEL
LIN {X 0,Y 278.656,Z 806.884,A -85,B 0,C 180,E1 19286.108,E2 19286.108} C_VEL
LIN {X 0,Y 281.003,Z 820.177,A -85,B 0,C 180,E1 19289.482,E2 19289.482} C_VEL
LIN {X 0,Y 264.553,Z 856.636,A -85,B 0,C 180,E1 19293.468,E2 19293.468} C_VEL
LIN {X 0,Y 247.832,Z 887.818,A -85,B 0,C 180,E1 19298.675,E2 19298.675} C_VEL
LIN {X 0,Y 232.445,Z 914.426,A -85,B 0,C 180,E1 19305.344,E2 19305.344} C_VEL
LIN {X 0,Y 219.596,Z 936.84,A -85,B 0,C 180,E1 19313.652,E2 19313.652} C_VEL
LIN {X 0,Y 210.713,Z 954.923,A -85,B 0,C 180,E1 19323.669,E2 19323.669} C_VEL
LIN {X 0,Y 207.489,Z 966.092,A -85,B 0,C 180,E1 19333.088,E2 19333.088} C_VEL
LIN {X 0,Y 207.253,Z 972.174,A -85,B 0,C 180,E1 19341.627,E2 19341.627} C_VEL
LIN {X 0,Y 208.035,Z 974.396,A -85,B 0,C 180,E1 19350,E2 19350} C_VEL
LIN {X 0,Y 207.244,Z 972.188,A -85,B 0,C 180,E1 19358.373,E2 19358.373} C_VEL
LIN {X 0,Y 207.741,Z 964.954,A -85,B 0,C 180,E1 19368.159,E2 19368.159} C_VEL
LIN {X 0,Y 212.611,Z 950.725,A -85,B 0,C 180,E1 19379.099,E2 19379.099} C_VEL
LIN {X 0,Y 223.05,Z 930.604,A -85,B 0,C 180,E1 19389.034,E2 19389.034} C_VEL
LIN {X 0,Y 237.234,Z 906.302,A -85,B 0,C 180,E1 19397.011,E2 19397.011} C_VEL
LIN {X 0,Y 253.526,Z 877.835,A -85,B 0,C 180,E1 19403.251,E2 19403.251} C_VEL
LIN {X 0,Y 270.394,Z 844.823,A -85,B 0,C 180,E1 19408.044,E2 19408.044} C_VEL
LIN {X 0,Y 281.128,Z 819.48,A -85,B 0,C 180,E1 19410.669,E2 19410.669} C_VEL
LIN {X 0,Y 277.074,Z 799.879,A -85,B 0,C 180,E1 19415.9,E2 19415.9} C_VEL
LIN {X 0,Y 271.01,Z 781.271,A -85,B 0,C 180,E1 19422.521,E2 19422.521} C_VEL
LIN {X 0,Y 265.096,Z 766.783,A -85,B 0,C 180,E1 19430.162,E2 19430.162} C_VEL
LIN {X 0,Y 262.578,Z 760.815,A -85,B 0,C 180,E1 19435.049,E2 19435.049} C_VEL
LIN {X 0,Y 259.997,Z 757.818,A -85,B 0,C 180,E1 19443.321,E2 19443.321} C_VEL
LIN {X 0,Y 260.249,Z 761.559,A -85,B 0,C 180,E1 19451.703,E2 19451.703} C_VEL
LIN {X 0,Y 261.913,Z 769.961,A -85,B 0,C 180,E1 19458.676,E2 19458.676} C_VEL
LIN {X 0,Y 261.604,Z 776.274,A -85,B 0,C 180,E1 19461.193,E2 19461.193} C_VEL
LIN {X 0,Y 259.885,Z 788.705,A -85,B 0,C 180,E1 19465.225,E2 19465.225} C_VEL
LIN {X 0,Y 261.102,Z 803.904,A -85,B 0,C 180,E1 19471.9,E2 19471.9} C_VEL
LIN {X 0,Y 260.484,Z 819.76,A -85,B 0,C 180,E1 19477.772,E2 19477.772} C_VEL
LIN {X 0,Y 259.018,Z 827.67,A -85,B 0,C 180,E1 19480.387,E2 19480.387} C_VEL
LIN {X 0,Y 242.746,Z 852.707,A -85,B 0,C 180,E1 19486.215,E2 19486.215} C_VEL
LIN {X 0,Y 227.553,Z 872.886,A -85,B 0,C 180,E1 19493.357,E2 19493.357} C_VEL
LIN {X 0,Y 214.09,Z 889.387,A -85,B 0,C 180,E1 19502.733,E2 19502.733} C_VEL
LIN {X 0,Y 205.533,Z 899.672,A -85,B 0,C 180,E1 19512.922,E2 19512.922} C_VEL
LIN {X 0,Y 202.161,Z 904.036,A -85,B 0,C 180,E1 19521.414,E2 19521.414} C_VEL
LIN {X 0,Y 201.182,Z 905.504,A -85,B 0,C 180,E1 19530,E2 19530} C_VEL
LIN {X 0,Y 202.194,Z 903.981,A -85,B 0,C 180,E1 19538.584,E2 19538.584} C_VEL
LIN {X 0,Y 206.722,Z 898.073,A -85,B 0,C 180,E1 19548.955,E2 19548.955} C_VEL
LIN {X 0,Y 216.422,Z 886.445,A -85,B 0,C 180,E1 19559.214,E2 19559.214} C_VEL
LIN {X 0,Y 230.073,Z 869.693,A -85,B 0,C 180,E1 19567.878,E2 19567.878} C_VEL
LIN {X 0,Y 246.15,Z 847.565,A -85,B 0,C 180,E1 19575.08,E2 19575.08} C_VEL
LIN {X 0,Y 259.682,Z 825.977,A -85,B 0,C 180,E1 19579.901,E2 19579.901} C_VEL
LIN {X 0,Y 261.044,Z 808.534,A -85,B 0,C 180,E1 19586.151,E2 19586.151} C_VEL
LIN {X 0,Y 260.246,Z 792.367,A -85,B 0,C 180,E1 19592.84,E2 19592.84} C_VEL
LIN {X 0,Y 258.522,Z 779.697,A -85,B 0,C 180,E1 19599.508,E2 19599.508} C_VEL
LIN {X 0,Y 257.038,Z 770.543,A -85,B 0,C 180,E1 19606.426,E2 19606.426} C_VEL
LIN {X 0,Y 256.712,Z 767.31,A -85,B 0,C 180,E1 19609.85,E2 19609.85} C_VEL
LIN {X 0,Y 256.96,Z 764.941,A -85,B 0,C 180,E1 19616.678,E2 19616.678} C_VEL
LIN {X 0,Y 258.698,Z 767.107,A -85,B 0,C 180,E1 19623.35,E2 19623.35} C_VEL
LIN {X 0,Y 261.452,Z 773.217,A -85,B 0,C 180,E1 19629.138,E2 19629.138} C_VEL
LIN {X 0,Y 266.44,Z 786.277,A -85,B 0,C 180,E1 19636.455,E2 19636.455} C_VEL
LIN {X 0,Y 271.876,Z 804.859,A -85,B 0,C 180,E1 19643.299,E2 19643.299} C_VEL
LIN {X 0,Y 275.253,Z 822.472,A -85,B 0,C 180,E1 19648.301,E2 19648.301} C_VEL
LIN {X 0,Y 258.835,Z 857.557,A -85,B 0,C 180,E1 19652.291,E2 19652.291} C_VEL
LIN {X 0,Y 242.095,Z 887.44,A -85,B 0,C 180,E1 19657.372,E2 19657.372} C_VEL
LIN {X 0,Y 225.345,Z 914.994,A -85,B 0,C 180,E1 19664.487,E2 19664.487} C_VEL
LIN {X 0,Y 211.083,Z 938.7,A -85,B 0,C 180,E1 19673.859,E2 19673.859} C_VEL
LIN {X 0,Y 202.274,Z 956.215,A -85,B 0,C 180,E1 19684.598,E2 19684.598} C_VEL
LIN {X 0,Y 199.44,Z 966.636,A -85,B 0,C 180,E1 19694.644,E2 19694.644} C_VEL
LIN {X 0,Y 199.397,Z 970.836,A -85,B 0,C 180,E1 19701.295,E2 19701.295} C_VEL
LIN {X 0,Y 200.235,Z 973.083,A -85,B 0,C 180,E1 19710,E2 19710} C_VEL
LIN {X 0,Y 199.391,Z 970.851,A -85,B 0,C 180,E1 19718.706,E2 19718.706} C_VEL
LIN {X 0,Y 200.002,Z 963.578,A -85,B 0,C 180,E1 19728.888,E2 19728.888} C_VEL
LIN {X 0,Y 205.092,Z 949.955,A -85,B 0,C 180,E1 19739.835,E2 19739.835} C_VEL
LIN {X 0,Y 216.348,Z 929.606,A -85,B 0,C 180,E1 19750.255,E2 19750.255} C_VEL
LIN {X 0,Y 231.536,Z 904.999,A -85,B 0,C 180,E1 19758.484,E2 19758.484} C_VEL
LIN {X 0,Y 248.834,Z 876.079,A -85,B 0,C 180,E1 19764.833,E2 19764.833} C_VEL
LIN {X 0,Y 265.982,Z 843.655,A -85,B 0,C 180,E1 19769.5,E2 19769.5} C_VEL
LIN {X 0,Y 275.286,Z 822.037,A -85,B 0,C 180,E1 19771.842,E2 19771.842} C_VEL
LIN {X 0,Y 271.749,Z 803.491,A -85,B 0,C 180,E1 19777.121,E2 19777.121} C_VEL
LIN {X 0,Y 266.568,Z 786.433,A -85,B 0,C 180,E1 19783.553,E2 19783.553} C_VEL
LIN {X 0,Y 261.608,Z 773.393,A -85,B 0,C 180,E1 19790.867,E2 19790.867} C_VEL
LIN {X 0,Y 258.871,Z 767.305,A -85,B 0,C 180,E1 19796.652,E2 19796.652} C_VEL
LIN {X 0,Y 257.053,Z 765.297,A -85,B 0,C 180,E1 19803.661,E2 19803.661} C_VEL
LIN {X 0,Y 256.894,Z 767.563,A -85,B 0,C 180,E1 19810.142,E2 19810.142} C_VEL
LIN {X 0,Y 258.095,Z 776.616,A -85,B 0,C 180,E1 19818.249,E2 19818.249} C_VEL
LIN {X 0,Y 259.885,Z 788.705,A -85,B 0,C 180,E1 19825.225,E2 19825.225} C_VEL
LIN {X 0,Y 259.024,Z 795.928,A -85,B 0,C 180,E1 19827.637,E2 19827.637} C_VEL
LIN {X 0,Y 255.746,Z 809.492,A -85,B 0,C 180,E1 19831.494,E2 19831.494} C_VEL
LIN {X 0,Y 254.333,Z 825.683,A -85,B 0,C 180,E1 19837.722,E2 19837.722} C_VEL
LIN {X 0,Y 253.373,Z 830.115,A -85,B 0,C 180,E1 19839.265,E2 19839.265} C_VEL
LIN {X 0,Y 236.11,Z 855.482,A -85,B 0,C 180,E1 19845.331,E2 19845.331} C_VEL
LIN {X 0,Y 219.71,Z 876.21,A -85,B 0,C 180,E1 19853.061,E2 19853.061} C_VEL
LIN {X 0,Y 205.974,Z 892.018,A -85,B 0,C 180,E1 19862.788,E2 19862.788} C_VEL
LIN {X 0,Y 198.076,Z 900.986,A -85,B 0,C 180,E1 19872.258,E2 19872.258} C_VEL
LIN {X 0,Y 194.46,Z 905.348,A -85,B 0,C 180,E1 19881.072,E2 19881.072} C_VEL
LIN {X 0,Y 193.417,Z 906.811,A -85,B 0,C 180,E1 19890,E2 19890} C_VEL
LIN {X 0,Y 194.49,Z 905.293,A -85,B 0,C 180,E1 19898.927,E2 19898.927} C_VEL
LIN {X 0,Y 199.499,Z 899.221,A -85,B 0,C 180,E1 19909.9,E2 19909.9} C_VEL
LIN {X 0,Y 209.686,Z 887.705,A -85,B 0,C 180,E1 19920.303,E2 19920.303} C_VEL
LIN {X 0,Y 224.144,Z 870.773,A -85,B 0,C 180,E1 19929.212,E2 19929.212} C_VEL
LIN {X 0,Y 240.883,Z 848.679,A -85,B 0,C 180,E1 19936.456,E2 19936.456} C_VEL
LIN {X 0,Y 253.519,Z 829.688,A -85,B 0,C 180,E1 19940.695,E2 19940.695} C_VEL
LIN {X 0,Y 255.573,Z 812.758,A -85,B 0,C 180,E1 19947.049,E2 19947.049} C_VEL
LIN {X 0,Y 255.409,Z 797.311,A -85,B 0,C 180,E1 19953.765,E2 19953.765} C_VEL
LIN {X 0,Y 254.167,Z 784.62,A -85,B 0,C 180,E1 19960.951,E2 19960.951} C_VEL
LIN {X 0,Y 253.38,Z 776.192,A -85,B 0,C 180,E1 19967.977,E2 19967.977} C_VEL
LIN {X 0,Y 253.775,Z 772.217,A -85,B 0,C 180,E1 19976.598,E2 19976.598} C_VEL
LIN {X 0,Y 255.602,Z 774.427,A -85,B 0,C 180,E1 19983.391,E2 19983.391} C_VEL
LIN {X 0,Y 259.074,Z 783.3,A -85,B 0,C 180,E1 19990.918,E2 19990.918} C_VEL
LIN {X 0,Y 263.351,Z 796.223,A -85,B 0,C 180,E1 19997.512,E2 19997.512} C_VEL
LIN {X 0,Y 267.492,Z 813.033,A -85,B 0,C 180,E1 20003.581,E2 20003.581} C_VEL
LIN {X 0,Y 269.387,Z 826.001,A -85,B 0,C 180,E1 20007.309,E2 20007.309} C_VEL
LIN {X 0,Y 252.355,Z 860.095,A -85,B 0,C 180,E1 20011.288,E2 20011.288} C_VEL
LIN {X 0,Y 233.754,Z 891.573,A -85,B 0,C 180,E1 20016.978,E2 20016.978} C_VEL
LIN {X 0,Y 216.324,Z 918.596,A -85,B 0,C 180,E1 20024.629,E2 20024.629} C_VEL
LIN {X 0,Y 202.417,Z 940.428,A -85,B 0,C 180,E1 20034.156,E2 20034.156} C_VEL
LIN {X 0,Y 194.299,Z 956.189,A -85,B 0,C 180,E1 20044.713,E2 20044.713} C_VEL
LIN {X 0,Y 191.633,Z 965.268,A -85,B 0,C 180,E1 20054.002,E2 20054.002} C_VEL
LIN {X 0,Y 191.582,Z 969.504,A -85,B 0,C 180,E1 20060.936,E2 20060.936} C_VEL
LIN {X 0,Y 192.437,Z 971.77,A -85,B 0,C 180,E1 20070,E2 20070} C_VEL
LIN {X 0,Y 191.578,Z 969.519,A -85,B 0,C 180,E1 20079.064,E2 20079.064} C_VEL
LIN {X 0,Y 192.271,Z 962.243,A -85,B 0,C 180,E1 20089.631,E2 20089.631} C_VEL
LIN {X 0,Y 197.883,Z 948.63,A -85,B 0,C 180,E1 20100.98,E2 20100.98} C_VEL
LIN {X 0,Y 209.044,Z 929.765,A -85,B 0,C 180,E1 20111.065,E2 20111.065} C_VEL
LIN {X 0,Y 224.922,Z 905.389,A -85,B 0,C 180,E1 20119.561,E2 20119.561} C_VEL
LIN {X 0,Y 242.63,Z 877.171,A -85,B 0,C 180,E1 20125.957,E2 20125.957} C_VEL
LIN {X 0,Y 259.878,Z 846.108,A -85,B 0,C 180,E1 20130.573,E2 20130.573} C_VEL
LIN {X 0,Y 269.544,Z 824.983,A -85,B 0,C 180,E1 20132.94,E2 20132.94} C_VEL
LIN {X 0,Y 266.141,Z 805.869,A -85,B 0,C 180,E1 20138.805,E2 20138.805} C_VEL
LIN {X 0,Y 261.74,Z 790.639,A -85,B 0,C 180,E1 20145.093,E2 20145.093} C_VEL
LIN {X 0,Y 257.854,Z 779.885,A -85,B 0,C 180,E1 20151.581,E2 20151.581} C_VEL
LIN {X 0,Y 255.762,Z 774.628,A -85,B 0,C 180,E1 20156.611,E2 20156.611} C_VEL
LIN {X 0,Y 253.94,Z 772.461,A -85,B 0,C 180,E1 20163.4,E2 20163.4} C_VEL
LIN {X 0,Y 253.553,Z 774.971,A -85,B 0,C 180,E1 20170.277,E2 20170.277} C_VEL
LIN {X 0,Y 254.198,Z 783.73,A -85,B 0,C 180,E1 20178.231,E2 20178.231} C_VEL
LIN {X 0,Y 255.441,Z 796.543,A -85,B 0,C 180,E1 20185.654,E2 20185.654} C_VEL
LIN {X 0,Y 255.746,Z 809.492,A -85,B 0,C 180,E1 20191.494,E2 20191.494} C_VEL
LIN {X 0,Y 253.651,Z 817.385,A -85,B 0,C 180,E1 20193.813,E2 20193.813} C_VEL
LIN {X 0,Y 248.071,Z 831.249,A -85,B 0,C 180,E1 20197.566,E2 20197.566} C_VEL
LIN {X 0,Y 245.032,Z 836.918,A -85,B 0,C 180,E1 20198.969,E2 20198.969} C_VEL
LIN {X 0,Y 226.514,Z 862.052,A -85,B 0,C 180,E1 20205.614,E2 20205.614} C_VEL
LIN {X 0,Y 210.217,Z 881.203,A -85,B 0,C 180,E1 20213.686,E2 20213.686} C_VEL
LIN {X 0,Y 196.84,Z 895.7,A -85,B 0,C 180,E1 20223.845,E2 20223.845} C_VEL
LIN {X 0,Y 189.228,Z 903.81,A -85,B 0,C 180,E1 20234.037,E2 20234.037} C_VEL
LIN {X 0,Y 186.076,Z 907.713,A -85,B 0,C 180,E1 20245.349,E2 20245.349} C_VEL
LIN {X 0,Y 186.079,Z 907.684,A -85,B 0,C 180,E1 20254.651,E2 20254.651} C_VEL
LIN {X 0,Y 189.285,Z 903.688,A -85,B 0,C 180,E1 20266.015,E2 20266.015} C_VEL
LIN {X 0,Y 198.019,Z 894.344,A -85,B 0,C 180,E1 20277.208,E2 20277.208} C_VEL
LIN {X 0,Y 211.963,Z 879.192,A -85,B 0,C 180,E1 20287.238,E2 20287.238} C_VEL
LIN {X 0,Y 228.634,Z 859.241,A -85,B 0,C 180,E1 20295.195,E2 20295.195} C_VEL
LIN {X 0,Y 246.313,Z 834.689,A -85,B 0,C 180,E1 20301.362,E2 20301.362} C_VEL
LIN {X 0,Y 248.146,Z 830.545,A -85,B 0,C 180,E1 20302.559,E2 20302.559} C_VEL
LIN {X 0,Y 250.272,Z 814.545,A -85,B 0,C 180,E1 20308.98,E2 20308.98} C_VEL
LIN {X 0,Y 250.432,Z 799.891,A -85,B 0,C 180,E1 20315.972,E2 20315.972} C_VEL
LIN {X 0,Y 249.847,Z 788.444,A -85,B 0,C 180,E1 20323.338,E2 20323.338} C_VEL
LIN {X 0,Y 249.814,Z 782.015,A -85,B 0,C 180,E1 20329.567,E2 20329.567} C_VEL
LIN {X 0,Y 250.465,Z 779.418,A -85,B 0,C 180,E1 20336.553,E2 20336.553} C_VEL
LIN {X 0,Y 251.317,Z 779.845,A -85,B 0,C 180,E1 20340.007,E2 20340.007} C_VEL
LIN {X 0,Y 253.208,Z 784.165,A -85,B 0,C 180,E1 20345.992,E2 20345.992} C_VEL
LIN {X 0,Y 256.447,Z 793.695,A -85,B 0,C 180,E1 20352.753,E2 20352.753} C_VEL
LIN {X 0,Y 260.215,Z 807.524,A -85,B 0,C 180,E1 20359.132,E2 20359.132} C_VEL
LIN {X 0,Y 263.346,Z 825.09,A -85,B 0,C 180,E1 20365.083,E2 20365.083} C_VEL
LIN {X 0,Y 263.378,Z 829.593,A -85,B 0,C 180,E1 20366.223,E2 20366.223} C_VEL
LIN {X 0,Y 245.074,Z 863.962,A -85,B 0,C 180,E1 20370.456,E2 20370.456} C_VEL
LIN {X 0,Y 226.567,Z 893.571,A -85,B 0,C 180,E1 20376.142,E2 20376.142} C_VEL
LIN {X 0,Y 209.039,Z 919.303,A -85,B 0,C 180,E1 20383.791,E2 20383.791} C_VEL
LIN {X 0,Y 194.455,Z 940.996,A -85,B 0,C 180,E1 20393.844,E2 20393.844} C_VEL
LIN {X 0,Y 185.732,Z 957.485,A -85,B 0,C 180,E1 20406.032,E2 20406.032} C_VEL
LIN {X 0,Y 183.602,Z 967.028,A -85,B 0,C 180,E1 20418.145,E2 20418.145} C_VEL
LIN {X 0,Y 184.064,Z 969.803,A -85,B 0,C 180,E1 20425.297,E2 20425.297} C_VEL
LIN {X 0,Y 184.633,Z 970.456,A -85,B 0,C 180,E1 20430,E2 20430} C_VEL
LIN {X 0,Y 183.719,Z 968.069,A -85,B 0,C 180,E1 20439.696,E2 20439.696} C_VEL
LIN {X 0,Y 184.609,Z 960.868,A -85,B 0,C 180,E1 20450.482,E2 20450.482} C_VEL
LIN {X 0,Y 190.787,Z 947.22,A -85,B 0,C 180,E1 20462.268,E2 20462.268} C_VEL
LIN {X 0,Y 202.978,Z 928.107,A -85,B 0,C 180,E1 20472.717,E2 20472.717} C_VEL
LIN {X 0,Y 219.593,Z 904.013,A -85,B 0,C 180,E1 20481.193,E2 20481.193} C_VEL
LIN {X 0,Y 238.107,Z 875.716,A -85,B 0,C 180,E1 20487.603,E2 20487.603} C_VEL
LIN {X 0,Y 255.956,Z 844.607,A -85,B 0,C 180,E1 20492.169,E2 20492.169} C_VEL
LIN {X 0,Y 263.878,Z 828.137,A -85,B 0,C 180,E1 20494.043,E2 20494.043} C_VEL
LIN {X 0,Y 261.114,Z 810.583,A -85,B 0,C 180,E1 20499.707,E2 20499.707} C_VEL
LIN {X 0,Y 257.08,Z 795.353,A -85,B 0,C 180,E1 20506.415,E2 20506.415} C_VEL
LIN {X 0,Y 253.66,Z 785.342,A -85,B 0,C 180,E1 20513.161,E2 20513.161} C_VEL
LIN {X 0,Y 252.509,Z 781.912,A -85,B 0,C 180,E1 20516.568,E2 20516.568} C_VEL
LIN {X 0,Y 250.609,Z 779.676,A -85,B 0,C 180,E1 20523.445,E2 20523.445} C_VEL
LIN {X 0,Y 249.968,Z 782.293,A -85,B 0,C 180,E1 20530.426,E2 20530.426} C_VEL
LIN {X 0,Y 250.103,Z 789.886,A -85,B 0,C 180,E1 20537.55,E2 20537.55} C_VEL
LIN {X 0,Y 250.561,Z 801.929,A -85,B 0,C 180,E1 20544.925,E2 20544.925} C_VEL
LIN {X 0,Y 250.173,Z 817.086,A -85,B 0,C 180,E1 20551.968,E2 20551.968} C_VEL
LIN {X 0,Y 248.071,Z 831.249,A -85,B 0,C 180,E1 20557.566,E2 20557.566} C_VEL
LIN {X 0,Y 244.486,Z 837.495,A -85,B 0,C 180,E1 20559.023,E2 20559.023} C_VEL
LIN {X 0,Y 228.506,Z 854.202,A -85,B 0,C 180,E1 20561.385,E2 20561.385} C_VEL
LIN {X 0,Y 227.938,Z 854.863,A -85,B 0,C 180,E1 20561.57,E2 20561.57} C_VEL
LIN {X 0,Y 210.342,Z 875.631,A -85,B 0,C 180,E1 20568.949,E2 20568.949} C_VEL
LIN {X 0,Y 194.924,Z 891.829,A -85,B 0,C 180,E1 20578.358,E2 20578.358} C_VEL
LIN {X 0,Y 184.834,Z 901.962,A -85,B 0,C 180,E1 20588.446,E2 20588.446} C_VEL
LIN {X 0,Y 179.074,Z 907.971,A -85,B 0,C 180,E1 20600.298,E2 20600.298} C_VEL
LIN {X 0,Y 177.872,Z 909.428,A -85,B 0,C 180,E1 20610,E2 20610} C_VEL
LIN {X 0,Y 179.102,Z 907.919,A -85,B 0,C 180,E1 20619.701,E2 20619.701} C_VEL
LIN {X 0,Y 184.875,Z 901.855,A -85,B 0,C 180,E1 20631.549,E2 20631.549} C_VEL
LIN {X 0,Y 196.268,Z 890.411,A -85,B 0,C 180,E1 20642.561,E2 20642.561} C_VEL
LIN {X 0,Y 212.089,Z 873.657,A -85,B 0,C 180,E1 20651.792,E2 20651.792} C_VEL
LIN {X 0,Y 230.109,Z 851.815,A -85,B 0,C 180,E1 20659.149,E2 20659.149} C_VEL
LIN {X 0,Y 241.766,Z 835.695,A -85,B 0,C 180,E1 20662.882,E2 20662.882} C_VEL
LIN {X 0,Y 244.655,Z 820.547,A -85,B 0,C 180,E1 20669.16,E2 20669.16} C_VEL
LIN {X 0,Y 245.637,Z 807.529,A -85,B 0,C 180,E1 20675.512,E2 20675.512} C_VEL
LIN {X 0,Y 245.714,Z 795.721,A -85,B 0,C 180,E1 20683.048,E2 20683.048} C_VEL
LIN {X 0,Y 246.003,Z 789.203,A -85,B 0,C 180,E1 20689.404,E2 20689.404} C_VEL
LIN {X 0,Y 246.927,Z 786.54,A -85,B 0,C 180,E1 20696.503,E2 20696.503} C_VEL
LIN {X 0,Y 247.796,Z 786.921,A -85,B 0,C 180,E1 20700.007,E2 20700.007} C_VEL
LIN {X 0,Y 249.356,Z 790.435,A -85,B 0,C 180,E1 20705.214,E2 20705.214} C_VEL
LIN {X 0,Y 252.222,Z 799.745,A -85,B 0,C 180,E1 20712.093,E2 20712.093} C_VEL
LIN {X 0,Y 255.328,Z 812.547,A -85,B 0,C 180,E1 20718.257,E2 20718.257} C_VEL
LIN {X 0,Y 257.93,Z 830.627,A -85,B 0,C 180,E1 20724.64,E2 20724.64} C_VEL
LIN {X 0,Y 254.899,Z 837.837,A -85,B 0,C 180,E1 20725.599,E2 20725.599} C_VEL
LIN {X 0,Y 234.942,Z 872.232,A -85,B 0,C 180,E1 20730.341,E2 20730.341} C_VEL
LIN {X 0,Y 215.735,Z 900.742,A -85,B 0,C 180,E1 20736.606,E2 20736.606} C_VEL
LIN {X 0,Y 197.822,Z 925.404,A -85,B 0,C 180,E1 20745.123,E2 20745.123} C_VEL
LIN {X 0,Y 184.916,Z 943.998,A -85,B 0,C 180,E1 20755.164,E2 20755.164} C_VEL
LIN {X 0,Y 177.293,Z 958.433,A -85,B 0,C 180,E1 20767.48,E2 20767.48} C_VEL
LIN {X 0,Y 175.757,Z 965.675,A -85,B 0,C 180,E1 20777.605,E2 20777.605} C_VEL
LIN {X 0,Y 176.201,Z 968.475,A -85,B 0,C 180,E1 20785.087,E2 20785.087} C_VEL
LIN {X 0,Y 176.834,Z 969.143,A -85,B 0,C 180,E1 20790,E2 20790} C_VEL
LIN {X 0,Y 175.876,Z 966.839,A -85,B 0,C 180,E1 20799.881,E2 20799.881} C_VEL
LIN {X 0,Y 176.917,Z 959.63,A -85,B 0,C 180,E1 20811.254,E2 20811.254} C_VEL
LIN {X 0,Y 183.811,Z 945.814,A -85,B 0,C 180,E1 20823.651,E2 20823.651} C_VEL
LIN {X 0,Y 196.963,Z 926.694,A -85,B 0,C 180,E1 20834.354,E2 20834.354} C_VEL
LIN {X 0,Y 214.198,Z 902.931,A -85,B 0,C 180,E1 20842.833,E2 20842.833} C_VEL
LIN {X 0,Y 233.816,Z 874.211,A -85,B 0,C 180,E1 20849.321,E2 20849.321} C_VEL
LIN {X 0,Y 252.788,Z 842.084,A -85,B 0,C 180,E1 20853.935,E2 20853.935} C_VEL
LIN {X 0,Y 258.167,Z 831.249,A -85,B 0,C 180,E1 20855.172,E2 20855.172} C_VEL
LIN {X 0,Y 255.846,Z 814.252,A -85,B 0,C 180,E1 20861.064,E2 20861.064} C_VEL
LIN {X 0,Y 252.355,Z 799.89,A -85,B 0,C 180,E1 20867.914,E2 20867.914} C_VEL
LIN {X 0,Y 249.484,Z 790.662,A -85,B 0,C 180,E1 20874.788,E2 20874.788} C_VEL
LIN {X 0,Y 247.892,Z 787.249,A -85,B 0,C 180,E1 20879.993,E2 20879.993} C_VEL
LIN {X 0,Y 247.071,Z 786.795,A -85,B 0,C 180,E1 20883.495,E2 20883.495} C_VEL
LIN {X 0,Y 246.064,Z 789.96,A -85,B 0,C 180,E1 20891.127,E2 20891.127} C_VEL
LIN {X 0,Y 245.813,Z 797.264,A -85,B 0,C 180,E1 20897.866,E2 20897.866} C_VEL
LIN {X 0,Y 245.703,Z 808.462,A -85,B 0,C 180,E1 20904.814,E2 20904.814} C_VEL
LIN {X 0,Y 244.453,Z 823.447,A -85,B 0,C 180,E1 20911.955,E2 20911.955} C_VEL
LIN {X 0,Y 241.654,Z 836.104,A -85,B 0,C 180,E1 20917.083,E2 20917.083} C_VEL
LIN {X 0,Y 227.938,Z 854.863,A -85,B 0,C 180,E1 20921.57,E2 20921.57} C_VEL
LIN {X 0,Y 217.17,Z 865.374,A -85,B 0,C 180,E1 20923.919,E2 20923.919} C_VEL
LIN {X 0,Y 206.455,Z 874.958,A -85,B 0,C 180,E1 20926.606,E2 20926.606} C_VEL
LIN {X 0,Y 189.624,Z 891.907,A -85,B 0,C 180,E1 20936.148,E2 20936.148} C_VEL
LIN {X 0,Y 177.589,Z 903.277,A -85,B 0,C 180,E1 20947.519,E2 20947.519} C_VEL
LIN {X 0,Y 171.391,Z 909.284,A -85,B 0,C 180,E1 20959.858,E2 20959.858} C_VEL
LIN {X 0,Y 170.088,Z 910.738,A -85,B 0,C 180,E1 20970,E2 20970} C_VEL
LIN {X 0,Y 171.419,Z 909.232,A -85,B 0,C 180,E1 20980.14,E2 20980.14} C_VEL
LIN {X 0,Y 177.621,Z 903.174,A -85,B 0,C 180,E1 20992.476,E2 20992.476} C_VEL
LIN {X 0,Y 189.709,Z 891.736,A -85,B 0,C 180,E1 21003.835,E2 21003.835} C_VEL
LIN {X 0,Y 206.556,Z 874.74,A -85,B 0,C 180,E1 21013.342,E2 21013.342} C_VEL
LIN {X 0,Y 225.476,Z 852.686,A -85,B 0,C 180,E1 21020.771,E2 21020.771} C_VEL
LIN {X 0,Y 236.361,Z 837.801,A -85,B 0,C 180,E1 21024.381,E2 21024.381} C_VEL
LIN {X 0,Y 239.47,Z 823.426,A -85,B 0,C 180,E1 21030.754,E2 21030.754} C_VEL
LIN {X 0,Y 240.88,Z 810.037,A -85,B 0,C 180,E1 21037.931,E2 21037.931} C_VEL
LIN {X 0,Y 241.567,Z 799.701,A -85,B 0,C 180,E1 21045.539,E2 21045.539} C_VEL
LIN {X 0,Y 242.016,Z 796.356,A -85,B 0,C 180,E1 21049.227,E2 21049.227} C_VEL
LIN {X 0,Y 243.162,Z 793.516,A -85,B 0,C 180,E1 21056.449,E2 21056.449} C_VEL
LIN {X 0,Y 244.49,Z 794.929,A -85,B 0,C 180,E1 21061.775,E2 21061.775} C_VEL
LIN {X 0,Y 246.791,Z 801.716,A -85,B 0,C 180,E1 21068.799,E2 21068.799} C_VEL
LIN {X 0,Y 249.582,Z 813.553,A -85,B 0,C 180,E1 21075.613,E2 21075.613} C_VEL
LIN {X 0,Y 251.955,Z 830.062,A -85,B 0,C 180,E1 21082.209,E2 21082.209} C_VEL
LIN {X 0,Y 251.837,Z 835.571,A -85,B 0,C 180,E1 21083.838,E2 21083.838} C_VEL
LIN {X 0,Y 231.569,Z 869.747,A -85,B 0,C 180,E1 21088.392,E2 21088.392} C_VEL
LIN {X 0,Y 211.148,Z 898.967,A -85,B 0,C 180,E1 21094.702,E2 21094.702} C_VEL
LIN {X 0,Y 192.983,Z 922.792,A -85,B 0,C 180,E1 21102.856,E2 21102.856} C_VEL
LIN {X 0,Y 178.121,Z 942.583,A -85,B 0,C 180,E1 21113.628,E2 21113.628} C_VEL
LIN {X 0,Y 169.739,Z 957.048,A -85,B 0,C 180,E1 21126.418,E2 21126.418} C_VEL
LIN {X 0,Y 167.934,Z 964.325,A -85,B 0,C 180,E1 21137.018,E2 21137.018} C_VEL
LIN {X 0,Y 168.334,Z 967.145,A -85,B 0,C 180,E1 21144.857,E2 21144.857} C_VEL
LIN {X 0,Y 169.023,Z 967.828,A -85,B 0,C 180,E1 21150,E2 21150} C_VEL
LIN {X 0,Y 168.006,Z 965.494,A -85,B 0,C 180,E1 21160.349,E2 21160.349} C_VEL
LIN {X 0,Y 169.299,Z 958.247,A -85,B 0,C 180,E1 21172.26,E2 21172.26} C_VEL
LIN {X 0,Y 176.947,Z 944.408,A -85,B 0,C 180,E1 21185.144,E2 21185.144} C_VEL
LIN {X 0,Y 192.037,Z 924.078,A -85,B 0,C 180,E1 21196.623,E2 21196.623} C_VEL
LIN {X 0,Y 210.847,Z 899.409,A -85,B 0,C 180,E1 21205.227,E2 21205.227} C_VEL
LIN {X 0,Y 231.577,Z 869.923,A -85,B 0,C 180,E1 21211.604,E2 21211.604} C_VEL
LIN {X 0,Y 252.054,Z 835.523,A -85,B 0,C 180,E1 21216.173,E2 21216.173} C_VEL
LIN {X 0,Y 251.464,Z 823.674,A -85,B 0,C 180,E1 21220.126,E2 21220.126} C_VEL
LIN {X 0,Y 248.712,Z 808.866,A -85,B 0,C 180,E1 21226.843,E2 21226.843} C_VEL
LIN {X 0,Y 246.274,Z 799.709,A -85,B 0,C 180,E1 21232.955,E2 21232.955} C_VEL
LIN {X 0,Y 245.202,Z 796.197,A -85,B 0,C 180,E1 21236.465,E2 21236.465} C_VEL
LIN {X 0,Y 244.197,Z 794.232,A -85,B 0,C 180,E1 21239.993,E2 21239.993} C_VEL
LIN {X 0,Y 242.7,Z 794.387,A -85,B 0,C 180,E1 21245.844,E2 21245.844} C_VEL
LIN {X 0,Y 241.823,Z 798.255,A -85,B 0,C 180,E1 21252.607,E2 21252.607} C_VEL
LIN {X 0,Y 241.156,Z 807.372,A -85,B 0,C 180,E1 21260.182,E2 21260.182} C_VEL
LIN {X 0,Y 239.98,Z 820.393,A -85,B 0,C 180,E1 21267.61,E2 21267.61} C_VEL
LIN {X 0,Y 237.211,Z 834.858,A -85,B 0,C 180,E1 21274.21,E2 21274.21} C_VEL
LIN {X 0,Y 236.13,Z 838.793,A -85,B 0,C 180,E1 21275.842,E2 21275.842} C_VEL
LIN {X 0,Y 216.758,Z 863.476,A -85,B 0,C 180,E1 21282.296,E2 21282.296} C_VEL
LIN {X 0,Y 206.455,Z 874.958,A -85,B 0,C 180,E1 21286.606,E2 21286.606} C_VEL
LIN {X 0,Y 195.778,Z 883.594,A -85,B 0,C 180,E1 21289.722,E2 21289.722} C_VEL
LIN {X 0,Y 185.421,Z 891.202,A -85,B 0,C 180,E1 21293.312,E2 21293.312} C_VEL
LIN {X 0,Y 172.5,Z 902.798,A -85,B 0,C 180,E1 21304.063,E2 21304.063} C_VEL
LIN {X 0,Y 165.601,Z 908.811,A -85,B 0,C 180,E1 21314.135,E2 21314.135} C_VEL
LIN {X 0,Y 162.803,Z 911.645,A -85,B 0,C 180,E1 21324.682,E2 21324.682} C_VEL
LIN {X 0,Y 162.808,Z 911.617,A -85,B 0,C 180,E1 21335.318,E2 21335.318} C_VEL
LIN {X 0,Y 167.458,Z 907.108,A -85,B 0,C 180,E1 21349.221,E2 21349.221} C_VEL
LIN {X 0,Y 178.686,Z 897.214,A -85,B 0,C 180,E1 21361.737,E2 21361.737} C_VEL
LIN {X 0,Y 195.727,Z 881.289,A -85,B 0,C 180,E1 21372.423,E2 21372.423} C_VEL
LIN {X 0,Y 215.108,Z 860.548,A -85,B 0,C 180,E1 21380.503,E2 21380.503} C_VEL
LIN {X 0,Y 230.034,Z 842.094,A -85,B 0,C 180,E1 21385.187,E2 21385.187} C_VEL
LIN {X 0,Y 233.749,Z 829.187,A -85,B 0,C 180,E1 21391.005,E2 21391.005} C_VEL
LIN {X 0,Y 235.93,Z 815.816,A -85,B 0,C 180,E1 21398.438,E2 21398.438} C_VEL
LIN {X 0,Y 237.115,Z 806.814,A -85,B 0,C 180,E1 21405.261,E2 21405.261} C_VEL
LIN {X 0,Y 237.773,Z 803.365,A -85,B 0,C 180,E1 21409.032,E2 21409.032} C_VEL
LIN {X 0,Y 239.251,Z 800.449,A -85,B 0,C 180,E1 21416.391,E2 21416.391} C_VEL
LIN {X 0,Y 240.637,Z 801.868,A -85,B 0,C 180,E1 21421.803,E2 21421.803} C_VEL
LIN {X 0,Y 242.721,Z 808.915,A -85,B 0,C 180,E1 21428.948,E2 21428.948} C_VEL
LIN {X 0,Y 244.847,Z 819.602,A -85,B 0,C 180,E1 21435.19,E2 21435.19} C_VEL
LIN {X 0,Y 246.646,Z 836.045,A -85,B 0,C 180,E1 21441.931,E2 21441.931} C_VEL
LIN {X 0,Y 245.418,Z 839.847,A -85,B 0,C 180,E1 21442.735,E2 21442.735} C_VEL
LIN {X 0,Y 224.951,Z 872.348,A -85,B 0,C 180,E1 21447.275,E2 21447.275} C_VEL
LIN {X 0,Y 204.462,Z 900.154,A -85,B 0,C 180,E1 21453.528,E2 21453.528} C_VEL
LIN {X 0,Y 184.452,Z 924.968,A -85,B 0,C 180,E1 21462.584,E2 21462.584} C_VEL
LIN {X 0,Y 168.702,Z 945.061,A -85,B 0,C 180,E1 21474.901,E2 21474.901} C_VEL
LIN {X 0,Y 161.316,Z 957.848,A -85,B 0,C 180,E1 21488.027,E2 21488.027} C_VEL
LIN {X 0,Y 160.136,Z 964.127,A -85,B 0,C 180,E1 21499.137,E2 21499.137} C_VEL
LIN {X 0,Y 161.226,Z 966.516,A -85,B 0,C 180,E1 21510,E2 21510} C_VEL
LIN {X 0,Y 160.147,Z 964.148,A -85,B 0,C 180,E1 21520.862,E2 21520.862} C_VEL
LIN {X 0,Y 161.745,Z 956.866,A -85,B 0,C 180,E1 21533.36,E2 21533.36} C_VEL
LIN {X 0,Y 169.679,Z 943.775,A -85,B 0,C 180,E1 21546.192,E2 21546.192} C_VEL
LIN {X 0,Y 186.016,Z 923.124,A -85,B 0,C 180,E1 21558.284,E2 21558.284} C_VEL
LIN {X 0,Y 205.316,Z 899.12,A -85,B 0,C 180,E1 21566.81,E2 21566.81} C_VEL
LIN {X 0,Y 226.357,Z 870.501,A -85,B 0,C 180,E1 21573.079,E2 21573.079} C_VEL
LIN {X 0,Y 246.406,Z 838.414,A -85,B 0,C 180,E1 21577.444,E2 21577.444} C_VEL
LIN {X 0,Y 246.117,Z 827.726,A -85,B 0,C 180,E1 21581.217,E2 21581.217} C_VEL
LIN {X 0,Y 244.031,Z 814.623,A -85,B 0,C 180,E1 21587.495,E2 21587.495} C_VEL
LIN {X 0,Y 241.762,Z 804.905,A -85,B 0,C 180,E1 21594.621,E2 21594.621} C_VEL
LIN {X 0,Y 240.357,Z 801.141,A -85,B 0,C 180,E1 21599.993,E2 21599.993} C_VEL
LIN {X 0,Y 239.367,Z 800.694,A -85,B 0,C 180,E1 21603.607,E2 21603.607} C_VEL
LIN {X 0,Y 237.877,Z 803.669,A -85,B 0,C 180,E1 21610.963,E2 21610.963} C_VEL
LIN {X 0,Y 236.604,Z 811.846,A -85,B 0,C 180,E1 21618.587,E2 21618.587} C_VEL
LIN {X 0,Y 234.932,Z 823.601,A -85,B 0,C 180,E1 21625.943,E2 21625.943} C_VEL
LIN {X 0,Y 232.06,Z 836.507,A -85,B 0,C 180,E1 21632.292,E2 21632.292} C_VEL
LIN {X 0,Y 229.915,Z 842.481,A -85,B 0,C 180,E1 21634.784,E2 21634.784} C_VEL
LIN {X 0,Y 210.42,Z 866.054,A -85,B 0,C 180,E1 21641.15,E2 21641.15} C_VEL
LIN {X 0,Y 191.767,Z 885.216,A -85,B 0,C 180,E1 21649.551,E2 21649.551} C_VEL
LIN {X 0,Y 185.421,Z 891.202,A -85,B 0,C 180,E1 21653.312,E2 21653.312} C_VEL
LIN {X 0,Y 175.494,Z 897.864,A -85,B 0,C 180,E1 21657.391,E2 21657.391} C_VEL
LIN {X 0,Y 166.273,Z 903.435,A -85,B 0,C 180,E1 21662.035,E2 21662.035} C_VEL
LIN {X 0,Y 158.096,Z 910.126,A -85,B 0,C 180,E1 21673.361,E2 21673.361} C_VEL
LIN {X 0,Y 155.058,Z 912.955,A -85,B 0,C 180,E1 21684.415,E2 21684.415} C_VEL
LIN {X 0,Y 155.064,Z 912.927,A -85,B 0,C 180,E1 21695.585,E2 21695.585} C_VEL
LIN {X 0,Y 159.182,Z 909.215,A -85,B 0,C 180,E1 21708.609,E2 21708.609} C_VEL
LIN {X 0,Y 170.741,Z 899.637,A -85,B 0,C 180,E1 21722.024,E2 21722.024} C_VEL
LIN {X 0,Y 188.012,Z 884.497,A -85,B 0,C 180,E1 21733.017,E2 21733.017} C_VEL
LIN {X 0,Y 209.019,Z 863.261,A -85,B 0,C 180,E1 21741.731,E2 21741.731} C_VEL
LIN {X 0,Y 225.002,Z 844.102,A -85,B 0,C 180,E1 21746.766,E2 21746.766} C_VEL
LIN {X 0,Y 228.944,Z 830.847,A -85,B 0,C 180,E1 21753.381,E2 21753.381} C_VEL
LIN {X 0,Y 231.176,Z 820.469,A -85,B 0,C 180,E1 21759.708,E2 21759.708} C_VEL
LIN {X 0,Y 232.769,Z 812.291,A -85,B 0,C 180,E1 21766.512,E2 21766.512} C_VEL
LIN {X 0,Y 234.125,Z 808.215,A -85,B 0,C 180,E1 21772.926,E2 21772.926} C_VEL
LIN {X 0,Y 235.081,Z 807.227,A -85,B 0,C 180,E1 21776.327,E2 21776.327} C_VEL
LIN {X 0,Y 236.51,Z 808.639,A -85,B 0,C 180,E1 21781.835,E2 21781.835} C_VEL
LIN {X 0,Y 238.174,Z 814.735,A -85,B 0,C 180,E1 21788.202,E2 21788.202} C_VEL
LIN {X 0,Y 240.043,Z 826.542,A -85,B 0,C 180,E1 21795.262,E2 21795.262} C_VEL
LIN {X 0,Y 240.965,Z 839.814,A -85,B 0,C 180,E1 21800.879,E2 21800.879} C_VEL
LIN {X 0,Y 237.47,Z 846.66,A -85,B 0,C 180,E1 21801.893,E2 21801.893} C_VEL
LIN {X 0,Y 216.471,Z 877.554,A -85,B 0,C 180,E1 21806.585,E2 21806.585} C_VEL
LIN {X 0,Y 194.513,Z 905.268,A -85,B 0,C 180,E1 21813.492,E2 21813.492} C_VEL
LIN {X 0,Y 175.438,Z 927.476,A -85,B 0,C 180,E1 21822.596,E2 21822.596} C_VEL
LIN {X 0,Y 160.885,Z 945.085,A -85,B 0,C 180,E1 21834.439,E2 21834.439} C_VEL
LIN {X 0,Y 153.228,Z 957.739,A -85,B 0,C 180,E1 21848.784,E2 21848.784} C_VEL
LIN {X 0,Y 152.3,Z 962.782,A -85,B 0,C 180,E1 21858.571,E2 21858.571} C_VEL
LIN {X 0,Y 153.408,Z 965.2,A -85,B 0,C 180,E1 21870,E2 21870} C_VEL
LIN {X 0,Y 152.311,Z 962.803,A -85,B 0,C 180,E1 21881.429,E2 21881.429} C_VEL
LIN {X 0,Y 154.252,Z 955.484,A -85,B 0,C 180,E1 21894.567,E2 21894.567} C_VEL
LIN {X 0,Y 163.883,Z 941.239,A -85,B 0,C 180,E1 21908.767,E2 21908.767} C_VEL
LIN {X 0,Y 180.477,Z 921.845,A -85,B 0,C 180,E1 21920.191,E2 21920.191} C_VEL
LIN {X 0,Y 200.498,Z 898.191,A -85,B 0,C 180,E1 21928.651,E2 21928.651} C_VEL
LIN {X 0,Y 222.746,Z 869.05,A -85,B 0,C 180,E1 21934.97,E2 21934.97} C_VEL
LIN {X 0,Y 241.222,Z 840.336,A -85,B 0,C 180,E1 21938.913,E2 21938.913} C_VEL
LIN {X 0,Y 240.028,Z 825.251,A -85,B 0,C 180,E1 21945.43,E2 21945.43} C_VEL
LIN {X 0,Y 238.057,Z 813.753,A -85,B 0,C 180,E1 21952.71,E2 21952.71} C_VEL
LIN {X 0,Y 236.597,Z 808.907,A -85,B 0,C 180,E1 21958.166,E2 21958.166} C_VEL
LIN {X 0,Y 235.204,Z 807.465,A -85,B 0,C 180,E1 21963.671,E2 21963.671} C_VEL
LIN {X 0,Y 233.38,Z 810.589,A -85,B 0,C 180,E1 21971.177,E2 21971.177} C_VEL
LIN {X 0,Y 231.91,Z 816.987,A -85,B 0,C 180,E1 21977.484,E2 21977.484} C_VEL
LIN {X 0,Y 229.766,Z 828.086,A -85,B 0,C 180,E1 21984.871,E2 21984.871} C_VEL
LIN {X 0,Y 226.403,Z 840.335,A -85,B 0,C 180,E1 21991.28,E2 21991.28} C_VEL
LIN {X 0,Y 223.865,Z 845.972,A -85,B 0,C 180,E1 21993.629,E2 21993.629} C_VEL
LIN {X 0,Y 203.019,Z 869.869,A -85,B 0,C 180,E1 22000.372,E2 22000.372} C_VEL
LIN {X 0,Y 184.04,Z 888.288,A -85,B 0,C 180,E1 22009.009,E2 22009.009} C_VEL
LIN {X 0,Y 167.932,Z 902.075,A -85,B 0,C 180,E1 22020.382,E2 22020.382} C_VEL
LIN {X 0,Y 166.273,Z 903.435,A -85,B 0,C 180,E1 22022.035,E2 22022.035} C_VEL
LIN {X 0,Y 157.908,Z 908.128,A -85,B 0,C 180,E1 22027.217,E2 22027.217} C_VEL
LIN {X 0,Y 150.389,Z 911.588,A -85,B 0,C 180,E1 22032.981,E2 22032.981} C_VEL
LIN {X 0,Y 147.303,Z 914.267,A -85,B 0,C 180,E1 22044.12,E2 22044.12} C_VEL
LIN {X 0,Y 147.31,Z 914.239,A -85,B 0,C 180,E1 22055.88,E2 22055.88} C_VEL
LIN {X 0,Y 151.789,Z 910.533,A -85,B 0,C 180,E1 22069.552,E2 22069.552} C_VEL
LIN {X 0,Y 164.153,Z 900.959,A -85,B 0,C 180,E1 22083.474,E2 22083.474} C_VEL
LIN {X 0,Y 181.78,Z 886.324,A -85,B 0,C 180,E1 22094.412,E2 22094.412} C_VEL
LIN {X 0,Y 203.037,Z 865.967,A -85,B 0,C 180,E1 22103.03,E2 22103.03} C_VEL
LIN {X 0,Y 219.475,Z 847.051,A -85,B 0,C 180,E1 22108.145,E2 22108.145} C_VEL
LIN {X 0,Y 223.758,Z 834.714,A -85,B 0,C 180,E1 22114.71,E2 22114.71} C_VEL
LIN {X 0,Y 226.463,Z 824.654,A -85,B 0,C 180,E1 22121.338,E2 22121.338} C_VEL
LIN {X 0,Y 228.68,Z 817.088,A -85,B 0,C 180,E1 22128.59,E2 22128.59} C_VEL
LIN {X 0,Y 230.728,Z 813.904,A -85,B 0,C 180,E1 22136.258,E2 22136.258} C_VEL
LIN {X 0,Y 232.251,Z 815.345,A -85,B 0,C 180,E1 22141.869,E2 22141.869} C_VEL
LIN {X 0,Y 233.668,Z 821.662,A -85,B 0,C 180,E1 22148.361,E2 22148.361} C_VEL
LIN {X 0,Y 235.012,Z 832.482,A -85,B 0,C 180,E1 22154.889,E2 22154.889} C_VEL
LIN {X 0,Y 235,Z 844.44,A -85,B 0,C 180,E1 22159.947,E2 22159.947} C_VEL
LIN {X 0,Y 212.131,Z 877.104,A -85,B 0,C 180,E1 22164.793,E2 22164.793} C_VEL
LIN {X 0,Y 190.072,Z 903.847,A -85,B 0,C 180,E1 22171.411,E2 22171.411} C_VEL
LIN {X 0,Y 169.449,Z 926.575,A -85,B 0,C 180,E1 22180.804,E2 22180.804} C_VEL
LIN {X 0,Y 153.191,Z 944.933,A -85,B 0,C 180,E1 22193.77,E2 22193.77} C_VEL
LIN {X 0,Y 145.255,Z 957.39,A -85,B 0,C 180,E1 22209.244,E2 22209.244} C_VEL
LIN {X 0,Y 144.445,Z 961.43,A -85,B 0,C 180,E1 22217.94,E2 22217.94} C_VEL
LIN {X 0,Y 145.573,Z 963.88,A -85,B 0,C 180,E1 22230,E2 22230} C_VEL
LIN {X 0,Y 144.459,Z 961.453,A -85,B 0,C 180,E1 22242.059,E2 22242.059} C_VEL
LIN {X 0,Y 146.835,Z 954.102,A -85,B 0,C 180,E1 22255.897,E2 22255.897} C_VEL
LIN {X 0,Y 157.182,Z 940.204,A -85,B 0,C 180,E1 22270.377,E2 22270.377} C_VEL
LIN {X 0,Y 174.696,Z 921.045,A -85,B 0,C 180,E1 22282.005,E2 22282.005} C_VEL
LIN {X 0,Y 196.605,Z 896.413,A -85,B 0,C 180,E1 22290.816,E2 22290.816} C_VEL
LIN {X 0,Y 219.399,Z 867.606,A -85,B 0,C 180,E1 22296.913,E2 22296.913} C_VEL
LIN {X 0,Y 235.625,Z 843.2,A -85,B 0,C 180,E1 22300.347,E2 22300.347} C_VEL
LIN {X 0,Y 234.851,Z 829.288,A -85,B 0,C 180,E1 22306.846,E2 22306.846} C_VEL
LIN {X 0,Y 233.616,Z 820.608,A -85,B 0,C 180,E1 22312.571,E2 22312.571} C_VEL
LIN {X 0,Y 232.322,Z 815.611,A -85,B 0,C 180,E1 22318.132,E2 22318.132} C_VEL
LIN {X 0,Y 230.848,Z 814.123,A -85,B 0,C 180,E1 22323.741,E2 22323.741} C_VEL
LIN {X 0,Y 228.747,Z 817.388,A -85,B 0,C 180,E1 22331.406,E2 22331.406} C_VEL
LIN {X 0,Y 226.528,Z 825.001,A -85,B 0,C 180,E1 22338.71,E2 22338.71} C_VEL
LIN {X 0,Y 223.456,Z 836.382,A -85,B 0,C 180,E1 22346.072,E2 22346.072} C_VEL
LIN {X 0,Y 219.433,Z 847.397,A -85,B 0,C 180,E1 22351.847,E2 22351.847} C_VEL
LIN {X 0,Y 198.051,Z 871.204,A -85,B 0,C 180,E1 22358.651,E2 22358.651} C_VEL
LIN {X 0,Y 178.192,Z 889.617,A -85,B 0,C 180,E1 22367.354,E2 22367.354} C_VEL
LIN {X 0,Y 161.163,Z 903.395,A -85,B 0,C 180,E1 22379.004,E2 22379.004} C_VEL
LIN {X 0,Y 150.389,Z 911.588,A -85,B 0,C 180,E1 22392.981,E2 22392.981} C_VEL
LIN {X 0,Y 144.243,Z 914.199,A -85,B 0,C 180,E1 22399.265,E2 22399.265} C_VEL
LIN {X 0,Y 139.16,Z 915.722,A -85,B 0,C 180,E1 22406.04,E2 22406.04} C_VEL
LIN {X 0,Y 139.572,Z 915.55,A -85,B 0,C 180,E1 22416.207,E2 22416.207} C_VEL
LIN {X 0,Y 144.757,Z 911.617,A -85,B 0,C 180,E1 22431.078,E2 22431.078} C_VEL
LIN {X 0,Y 157.667,Z 902.282,A -85,B 0,C 180,E1 22445.047,E2 22445.047} C_VEL
LIN {X 0,Y 176.244,Z 887.674,A -85,B 0,C 180,E1 22456.18,E2 22456.18} C_VEL
LIN {X 0,Y 198.342,Z 867.41,A -85,B 0,C 180,E1 22464.795,E2 22464.795} C_VEL
LIN {X 0,Y 214.152,Z 849.871,A -85,B 0,C 180,E1 22469.651,E2 22469.651} C_VEL
LIN {X 0,Y 218.778,Z 838.224,A -85,B 0,C 180,E1 22476.348,E2 22476.348} C_VEL
LIN {X 0,Y 221.918,Z 828.711,A -85,B 0,C 180,E1 22483.212,E2 22483.212} C_VEL
LIN {X 0,Y 223.788,Z 823.752,A -85,B 0,C 180,E1 22488.338,E2 22488.338} C_VEL
LIN {X 0,Y 226.24,Z 820.497,A -85,B 0,C 180,E1 22496.183,E2 22496.183} C_VEL
LIN {X 0,Y 227.769,Z 821.938,A -85,B 0,C 180,E1 22501.905,E2 22501.905} C_VEL
LIN {X 0,Y 229.056,Z 828.882,A -85,B 0,C 180,E1 22508.818,E2 22508.818} C_VEL
LIN {X 0,Y 229.772,Z 839.743,A -85,B 0,C 180,E1 22515.236,E2 22515.236} C_VEL
LIN {X 0,Y 229.761,Z 845.938,A -85,B 0,C 180,E1 22518.1,E2 22518.1} C_VEL
LIN {X 0,Y 226.939,Z 851.089,A -85,B 0,C 180,E1 22519.018,E2 22519.018} C_VEL
LIN {X 0,Y 202.998,Z 882.865,A -85,B 0,C 180,E1 22524.155,E2 22524.155} C_VEL
LIN {X 0,Y 179.089,Z 909.688,A -85,B 0,C 180,E1 22531.683,E2 22531.683} C_VEL
LIN {X 0,Y 158.827,Z 930.494,A -85,B 0,C 180,E1 22541.697,E2 22541.697} C_VEL
LIN {X 0,Y 144.103,Z 946.421,A -85,B 0,C 180,E1 22554.835,E2 22554.835} C_VEL
LIN {X 0,Y 137.131,Z 957.36,A -85,B 0,C 180,E1 22570.724,E2 22570.724} C_VEL
LIN {X 0,Y 136.89,Z 961.823,A -85,B 0,C 180,E1 22583.671,E2 22583.671} C_VEL
LIN {X 0,Y 137.747,Z 962.563,A -85,B 0,C 180,E1 22590,E2 22590} C_VEL
LIN {X 0,Y 136.622,Z 960.102,A -85,B 0,C 180,E1 22602.762,E2 22602.762} C_VEL
LIN {X 0,Y 140.114,Z 951.768,A -85,B 0,C 180,E1 22618.665,E2 22618.665} C_VEL
LIN {X 0,Y 152.623,Z 937.028,A -85,B 0,C 180,E1 22633.796,E2 22633.796} C_VEL
LIN {X 0,Y 171.993,Z 917.258,A -85,B 0,C 180,E1 22645.296,E2 22645.296} C_VEL
LIN {X 0,Y 195.535,Z 891.856,A -85,B 0,C 180,E1 22653.783,E2 22653.783} C_VEL
LIN {X 0,Y 219.917,Z 861.297,A -85,B 0,C 180,E1 22659.649,E2 22659.649} C_VEL
LIN {X 0,Y 229.148,Z 848.044,A -85,B 0,C 180,E1 22661.368,E2 22661.368} C_VEL
LIN {X 0,Y 230.031,Z 844.793,A -85,B 0,C 180,E1 22662.4,E2 22662.4} C_VEL
LIN {X 0,Y 229.534,Z 832.822,A -85,B 0,C 180,E1 22668.619,E2 22668.619} C_VEL
LIN {X 0,Y 228.604,Z 825.353,A -85,B 0,C 180,E1 22674.311,E2 22674.311} C_VEL
LIN {X 0,Y 227.503,Z 821.116,A -85,B 0,C 180,E1 22679.993,E2 22679.993} C_VEL
LIN {X 0,Y 226.363,Z 820.699,A -85,B 0,C 180,E1 22683.815,E2 22683.815} C_VEL
LIN {X 0,Y 223.843,Z 824.072,A -85,B 0,C 180,E1 22691.66,E2 22691.66} C_VEL
LIN {X 0,Y 221.229,Z 831.471,A -85,B 0,C 180,E1 22698.79,E2 22698.79} C_VEL
LIN {X 0,Y 217.646,Z 841.718,A -85,B 0,C 180,E1 22705.668,E2 22705.668} C_VEL
LIN {X 0,Y 214.093,Z 850.21,A -85,B 0,C 180,E1 22710.324,E2 22710.324} C_VEL
LIN {X 0,Y 191.972,Z 873.824,A -85,B 0,C 180,E1 22717.298,E2 22717.298} C_VEL
LIN {X 0,Y 170.461,Z 892.564,A -85,B 0,C 180,E1 22726.681,E2 22726.681} C_VEL
LIN {X 0,Y 153.058,Z 905.737,A -85,B 0,C 180,E1 22738.829,E2 22738.829} C_VEL
LIN {X 0,Y 142.815,Z 912.979,A -85,B 0,C 180,E1 22752.331,E2 22752.331} C_VEL
LIN {X 0,Y 139.16,Z 915.722,A -85,B 0,C 180,E1 22766.04,E2 22766.04} C_VEL
LIN {X 0,Y 136.45,Z 916.362,A -85,B 0,C 180,E1 22771.367,E2 22771.367} C_VEL
LIN {X 0,Y 132.407,Z 916.394,A -85,B 0,C 180,E1 22780.372,E2 22780.372} C_VEL
LIN {X 0,Y 132.457,Z 916.21,A -85,B 0,C 180,E1 22780.609,E2 22780.609} C_VEL
LIN {X 0,Y 139.84,Z 911.427,A -85,B 0,C 180,E1 22795.571,E2 22795.571} C_VEL
LIN {X 0,Y 155.05,Z 901.016,A -85,B 0,C 180,E1 22809.399,E2 22809.399} C_VEL
LIN {X 0,Y 176.307,Z 884.597,A -85,B 0,C 180,E1 22820.381,E2 22820.381} C_VEL
LIN {X 0,Y 198.096,Z 864.555,A -85,B 0,C 180,E1 22827.935,E2 22827.935} C_VEL
LIN {X 0,Y 208.818,Z 852.962,A -85,B 0,C 180,E1 22831.12,E2 22831.12} C_VEL
LIN {X 0,Y 214.075,Z 841.232,A -85,B 0,C 180,E1 22838.364,E2 22838.364} C_VEL
LIN {X 0,Y 217.811,Z 832.167,A -85,B 0,C 180,E1 22845.911,E2 22845.911} C_VEL
LIN {X 0,Y 220.338,Z 827.762,A -85,B 0,C 180,E1 22853.147,E2 22853.147} C_VEL
LIN {X 0,Y 221.473,Z 826.889,A -85,B 0,C 180,E1 22856.101,E2 22856.101} C_VEL
LIN {X 0,Y 222.768,Z 827.237,A -85,B 0,C 180,E1 22860.007,E2 22860.007} C_VEL
LIN {X 0,Y 223.833,Z 832.749,A -85,B 0,C 180,E1 22866.782,E2 22866.782} C_VEL
LIN {X 0,Y 224.378,Z 842.984,A -85,B 0,C 180,E1 22873.621,E2 22873.621} C_VEL
LIN {X 0,Y 224.174,Z 849.508,A -85,B 0,C 180,E1 22876.869,E2 22876.869} C_VEL
LIN {X 0,Y 201.54,Z 879.292,A -85,B 0,C 180,E1 22881.568,E2 22881.568} C_VEL
LIN {X 0,Y 175.771,Z 907.372,A -85,B 0,C 180,E1 22889.033,E2 22889.033} C_VEL
LIN {X 0,Y 152.949,Z 929.5,A -85,B 0,C 180,E1 22899.639,E2 22899.639} C_VEL
LIN {X 0,Y 137.387,Z 945.018,A -85,B 0,C 180,E1 22912.837,E2 22912.837} C_VEL
LIN {X 0,Y 129.478,Z 955.989,A -85,B 0,C 180,E1 22929.535,E2 22929.535} C_VEL
LIN {X 0,Y 128.977,Z 960.482,A -85,B 0,C 180,E1 22943.281,E2 22943.281} C_VEL
LIN {X 0,Y 129.903,Z 961.242,A -85,B 0,C 180,E1 22950,E2 22950} C_VEL
LIN {X 0,Y 128.789,Z 958.749,A -85,B 0,C 180,E1 22963.552,E2 22963.552} C_VEL
LIN {X 0,Y 132.825,Z 950.512,A -85,B 0,C 180,E1 22980.18,E2 22980.18} C_VEL
LIN {X 0,Y 146.723,Z 935.623,A -85,B 0,C 180,E1 22996.048,E2 22996.048} C_VEL
LIN {X 0,Y 168.12,Z 915.087,A -85,B 0,C 180,E1 23007.992,E2 23007.992} C_VEL
LIN {X 0,Y 193.501,Z 888.789,A -85,B 0,C 180,E1 23016.392,E2 23016.392} C_VEL
LIN {X 0,Y 217.812,Z 859.003,A -85,B 0,C 180,E1 23021.792,E2 23021.792} C_VEL
LIN {X 0,Y 224.398,Z 849.486,A -85,B 0,C 180,E1 23023.144,E2 23023.144} C_VEL
LIN {X 0,Y 224.35,Z 837.849,A -85,B 0,C 180,E1 23029.556,E2 23029.556} C_VEL
LIN {X 0,Y 223.502,Z 830.037,A -85,B 0,C 180,E1 23036.122,E2 23036.122} C_VEL
LIN {X 0,Y 222.817,Z 827.521,A -85,B 0,C 180,E1 23039.993,E2 23039.993} C_VEL
LIN {X 0,Y 221.582,Z 827.105,A -85,B 0,C 180,E1 23043.897,E2 23043.897} C_VEL
LIN {X 0,Y 219.452,Z 829.287,A -85,B 0,C 180,E1 23049.89,E2 23049.89} C_VEL
LIN {X 0,Y 216.487,Z 835.652,A -85,B 0,C 180,E1 23057.116,E2 23057.116} C_VEL
LIN {X 0,Y 212.498,Z 845.323,A -85,B 0,C 180,E1 23064.176,E2 23064.176} C_VEL
LIN {X 0,Y 208.801,Z 853.231,A -85,B 0,C 180,E1 23068.828,E2 23068.828} C_VEL
LIN {X 0,Y 186.108,Z 876.245,A -85,B 0,C 180,E1 23075.824,E2 23075.824} C_VEL
LIN {X 0,Y 164.842,Z 893.888,A -85,B 0,C 180,E1 23084.81,E2 23084.81} C_VEL
LIN {X 0,Y 146.406,Z 907.057,A -85,B 0,C 180,E1 23097.241,E2 23097.241} C_VEL
LIN {X 0,Y 135.822,Z 914.067,A -85,B 0,C 180,E1 23110.531,E2 23110.531} C_VEL
LIN {X 0,Y 131.389,Z 917.035,A -85,B 0,C 180,E1 23125.843,E2 23125.843} C_VEL
LIN {X 0,Y 132.457,Z 916.21,A -85,B 0,C 180,E1 23140.609,E2 23140.609} C_VEL
LIN {X 0,Y 131.238,Z 915.251,A -85,B 0,C 180,E1 23148.203,E2 23148.203} C_VEL
LIN {X 0,Y 131.886,Z 913.273,A -85,B 0,C 180,E1 23155.82,E2 23155.82} C_VEL
LIN {X 0,Y 146.686,Z 903.91,A -85,B 0,C 180,E1 23169.708,E2 23169.708} C_VEL
LIN {X 0,Y 169.036,Z 887.866,A -85,B 0,C 180,E1 23181.442,E2 23181.442} C_VEL
LIN {X 0,Y 192.664,Z 867.271,A -85,B 0,C 180,E1 23189.491,E2 23189.491} C_VEL
LIN {X 0,Y 202.688,Z 857.175,A -85,B 0,C 180,E1 23192.139,E2 23192.139} C_VEL
LIN {X 0,Y 207.491,Z 848.525,A -85,B 0,C 180,E1 23197.496,E2 23197.496} C_VEL
LIN {X 0,Y 211.738,Z 839.761,A -85,B 0,C 180,E1 23204.475,E2 23204.475} C_VEL
LIN {X 0,Y 214.964,Z 834.374,A -85,B 0,C 180,E1 23211.938,E2 23211.938} C_VEL
LIN {X 0,Y 216.563,Z 833.203,A -85,B 0,C 180,E1 23216.012,E2 23216.012} C_VEL
LIN {X 0,Y 217.976,Z 833.565,A -85,B 0,C 180,E1 23220.008,E2 23220.008} C_VEL
LIN {X 0,Y 218.826,Z 839.245,A -85,B 0,C 180,E1 23226.938,E2 23226.938} C_VEL
LIN {X 0,Y 218.86,Z 849.13,A -85,B 0,C 180,E1 23233.53,E2 23233.53} C_VEL
LIN {X 0,Y 218.624,Z 852.565,A -85,B 0,C 180,E1 23235.333,E2 23235.333} C_VEL
LIN {X 0,Y 195.043,Z 881.916,A -85,B 0,C 180,E1 23240.154,E2 23240.154} C_VEL
LIN {X 0,Y 169.825,Z 907.888,A -85,B 0,C 180,E1 23247.308,E2 23247.308} C_VEL
LIN {X 0,Y 147.295,Z 928.524,A -85,B 0,C 180,E1 23257.437,E2 23257.437} C_VEL
LIN {X 0,Y 129.502,Z 944.986,A -85,B 0,C 180,E1 23272.284,E2 23272.284} C_VEL
LIN {X 0,Y 121.856,Z 954.613,A -85,B 0,C 180,E1 23288.192,E2 23288.192} C_VEL
LIN {X 0,Y 121.091,Z 959.144,A -85,B 0,C 180,E1 23302.841,E2 23302.841} C_VEL
LIN {X 0,Y 122.064,Z 959.923,A -85,B 0,C 180,E1 23310,E2 23310} C_VEL
LIN {X 0,Y 120.96,Z 957.391,A -85,B 0,C 180,E1 23324.448,E2 23324.448} C_VEL
LIN {X 0,Y 125.289,Z 949.68,A -85,B 0,C 180,E1 23341.236,E2 23341.236} C_VEL
LIN {X 0,Y 139.136,Z 935.975,A -85,B 0,C 180,E1 23357.06,E2 23357.06} C_VEL
LIN {X 0,Y 161.076,Z 916.226,A -85,B 0,C 180,E1 23369.332,E2 23369.332} C_VEL
LIN {X 0,Y 185.765,Z 892.143,A -85,B 0,C 180,E1 23377.519,E2 23377.519} C_VEL
LIN {X 0,Y 210.944,Z 863.296,A -85,B 0,C 180,E1 23383.078,E2 23383.078} C_VEL
LIN {X 0,Y 218.848,Z 852.503,A -85,B 0,C 180,E1 23384.705,E2 23384.705} C_VEL
LIN {X 0,Y 219.009,Z 841.946,A -85,B 0,C 180,E1 23391.075,E2 23391.075} C_VEL
LIN {X 0,Y 218.609,Z 836.452,A -85,B 0,C 180,E1 23396.035,E2 23396.035} C_VEL
LIN {X 0,Y 218.016,Z 833.831,A -85,B 0,C 180,E1 23399.992,E2 23399.992} C_VEL
LIN {X 0,Y 216.652,Z 833.425,A -85,B 0,C 180,E1 23403.986,E2 23403.986} C_VEL
LIN {X 0,Y 214.396,Z 835.494,A -85,B 0,C 180,E1 23409.814,E2 23409.814} C_VEL
LIN {X 0,Y 211.233,Z 841.199,A -85,B 0,C 180,E1 23416.594,E2 23416.594} C_VEL
LIN {X 0,Y 206.492,Z 850.756,A -85,B 0,C 180,E1 23423.867,E2 23423.867} C_VEL
LIN {X 0,Y 202.615,Z 857.479,A -85,B 0,C 180,E1 23427.822,E2 23427.822} C_VEL
LIN {X 0,Y 179.012,Z 879.812,A -85,B 0,C 180,E1 23434.726,E2 23434.726} C_VEL
LIN {X 0,Y 157.196,Z 896.803,A -85,B 0,C 180,E1 23443.949,E2 23443.949} C_VEL
LIN {X 0,Y 138.34,Z 909.397,A -85,B 0,C 180,E1 23456.949,E2 23456.949} C_VEL
LIN {X 0,Y 127.601,Z 915.911,A -85,B 0,C 180,E1 23471.045,E2 23471.045} C_VEL
LIN {X 0,Y 124.094,Z 918.198,A -85,B 0,C 180,E1 23483.016,E2 23483.016} C_VEL
LIN {X 0,Y 124.103,Z 918.172,A -85,B 0,C 180,E1 23496.984,E2 23496.984} C_VEL
LIN {X 0,Y 131.886,Z 913.273,A -85,B 0,C 180,E1 23515.82,E2 23515.82} C_VEL
LIN {X 0,Y 134.314,Z 910.499,A -85,B 0,C 180,E1 23523.212,E2 23523.212} C_VEL
LIN {X 0,Y 138.492,Z 906.62,A -85,B 0,C 180,E1 23530.194,E2 23530.194} C_VEL
LIN {X 0,Y 159.217,Z 892.858,A -85,B 0,C 180,E1 23541.522,E2 23541.522} C_VEL
LIN {X 0,Y 183.832,Z 873.153,A -85,B 0,C 180,E1 23550.148,E2 23550.148} C_VEL
LIN {X 0,Y 197.643,Z 860.064,A -85,B 0,C 180,E1 23553.754,E2 23553.754} C_VEL
LIN {X 0,Y 203.124,Z 851.055,A -85,B 0,C 180,E1 23559.957,E2 23559.957} C_VEL
LIN {X 0,Y 207.701,Z 843.239,A -85,B 0,C 180,E1 23567.42,E2 23567.42} C_VEL
LIN {X 0,Y 210.276,Z 840.119,A -85,B 0,C 180,E1 23573.412,E2 23573.412} C_VEL
LIN {X 0,Y 212.953,Z 839.682,A -85,B 0,C 180,E1 23580.008,E2 23580.008} C_VEL
LIN {X 0,Y 213.602,Z 845.659,A -85,B 0,C 180,E1 23587.109,E2 23587.109} C_VEL
LIN {X 0,Y 213.04,Z 855.654,A -85,B 0,C 180,E1 23593.761,E2 23593.761} C_VEL
LIN {X 0,Y 208.157,Z 862.314,A -85,B 0,C 180,E1 23594.871,E2 23594.871} C_VEL
LIN {X 0,Y 183.285,Z 890.003,A -85,B 0,C 180,E1 23599.931,E2 23599.931} C_VEL
LIN {X 0,Y 157.728,Z 914.037,A -85,B 0,C 180,E1 23607.754,E2 23607.754} C_VEL
LIN {X 0,Y 133.606,Z 934.492,A -85,B 0,C 180,E1 23620.326,E2 23620.326} C_VEL
LIN {X 0,Y 118.222,Z 948.258,A -85,B 0,C 180,E1 23636.716,E2 23636.716} C_VEL
LIN {X 0,Y 113.145,Z 956.006,A -85,B 0,C 180,E1 23654.53,E2 23654.53} C_VEL
LIN {X 0,Y 114.242,Z 958.606,A -85,B 0,C 180,E1 23670,E2 23670} C_VEL
LIN {X 0,Y 113.164,Z 956.032,A -85,B 0,C 180,E1 23685.467,E2 23685.467} C_VEL
LIN {X 0,Y 118.297,Z 948.287,A -85,B 0,C 180,E1 23703.313,E2 23703.313} C_VEL
LIN {X 0,Y 133.585,Z 934.565,A -85,B 0,C 180,E1 23719.684,E2 23719.684} C_VEL
LIN {X 0,Y 157.741,Z 914.156,A -85,B 0,C 180,E1 23732.236,E2 23732.236} C_VEL
LIN {X 0,Y 183.493,Z 889.983,A -85,B 0,C 180,E1 23740.099,E2 23740.099} C_VEL
LIN {X 0,Y 209.887,Z 860.445,A -85,B 0,C 180,E1 23745.425,E2 23745.425} C_VEL
LIN {X 0,Y 213.247,Z 855.68,A -85,B 0,C 180,E1 23746.239,E2 23746.239} C_VEL
LIN {X 0,Y 213.722,Z 845.801,A -85,B 0,C 180,E1 23752.895,E2 23752.895} C_VEL
LIN {X 0,Y 212.979,Z 839.966,A -85,B 0,C 180,E1 23759.992,E2 23759.992} C_VEL
LIN {X 0,Y 211.577,Z 839.616,A -85,B 0,C 180,E1 23764.082,E2 23764.082} C_VEL
LIN {X 0,Y 208.947,Z 841.765,A -85,B 0,C 180,E1 23770.072,E2 23770.072} C_VEL
LIN {X 0,Y 205.153,Z 847.76,A -85,B 0,C 180,E1 23777.101,E2 23777.101} C_VEL
LIN {X 0,Y 199.355,Z 857.82,A -85,B 0,C 180,E1 23784.725,E2 23784.725} C_VEL
LIN {X 0,Y 197.592,Z 860.339,A -85,B 0,C 180,E1 23786.19,E2 23786.19} C_VEL
LIN {X 0,Y 173.312,Z 882.263,A -85,B 0,C 180,E1 23793.068,E2 23793.068} C_VEL
LIN {X 0,Y 149.577,Z 899.719,A -85,B 0,C 180,E1 23802.995,E2 23802.995} C_VEL
LIN {X 0,Y 131.854,Z 910.715,A -85,B 0,C 180,E1 23815.095,E2 23815.095} C_VEL
LIN {X 0,Y 121.19,Z 916.697,A -85,B 0,C 180,E1 23828.066,E2 23828.066} C_VEL
LIN {X 0,Y 116.346,Z 919.513,A -85,B 0,C 180,E1 23842.548,E2 23842.548} C_VEL
LIN {X 0,Y 116.355,Z 919.487,A -85,B 0,C 180,E1 23857.452,E2 23857.452} C_VEL
LIN {X 0,Y 124.634,Z 914.729,A -85,B 0,C 180,E1 23877.05,E2 23877.05} C_VEL
LIN {X 0,Y 138.492,Z 906.62,A -85,B 0,C 180,E1 23890.194,E2 23890.194} C_VEL
LIN {X 0,Y 144.299,Z 901.912,A -85,B 0,C 180,E1 23896.618,E2 23896.618} C_VEL
LIN {X 0,Y 151.389,Z 896.337,A -85,B 0,C 180,E1 23902.466,E2 23902.466} C_VEL
LIN {X 0,Y 177.549,Z 876.628,A -85,B 0,C 180,E1 23911.611,E2 23911.611} C_VEL
LIN {X 0,Y 192.287,Z 863.429,A -85,B 0,C 180,E1 23915.34,E2 23915.34} C_VEL
LIN {X 0,Y 197.564,Z 855.787,A -85,B 0,C 180,E1 23920.804,E2 23920.804} C_VEL
LIN {X 0,Y 201.884,Z 849.431,A -85,B 0,C 180,E1 23927.051,E2 23927.051} C_VEL
LIN {X 0,Y 205.006,Z 846.1,A -85,B 0,C 180,E1 23933.585,E2 23933.585} C_VEL
LIN {X 0,Y 207.779,Z 845.677,A -85,B 0,C 180,E1 23940.008,E2 23940.008} C_VEL
LIN {X 0,Y 208.172,Z 850.649,A -85,B 0,C 180,E1 23946.25,E2 23946.25} C_VEL
LIN {X 0,Y 207.564,Z 858.728,A -85,B 0,C 180,E1 23952.072,E2 23952.072} C_VEL
LIN {X 0,Y 205.063,Z 862.213,A -85,B 0,C 180,E1 23952.849,E2 23952.849} C_VEL
LIN {X 0,Y 178.982,Z 890.176,A -85,B 0,C 180,E1 23957.837,E2 23957.837} C_VEL
LIN {X 0,Y 151.167,Z 915.011,A -85,B 0,C 180,E1 23966.05,E2 23966.05} C_VEL
LIN {X 0,Y 126.211,Z 934.785,A -85,B 0,C 180,E1 23979,E2 23979} C_VEL
LIN {X 0,Y 110.052,Z 948.151,A -85,B 0,C 180,E1 23996.738,E2 23996.738} C_VEL
LIN {X 0,Y 105.374,Z 954.644,A -85,B 0,C 180,E1 24013.357,E2 24013.357} C_VEL
LIN {X 0,Y 106.387,Z 957.283,A -85,B 0,C 180,E1 24030,E2 24030} C_VEL
LIN {X 0,Y 105.392,Z 954.672,A -85,B 0,C 180,E1 24046.64,E2 24046.64} C_VEL
LIN {X 0,Y 111.496,Z 946.872,A -85,B 0,C 180,E1 24065.684,E2 24065.684} C_VEL
LIN {X 0,Y 128.343,Z 933.156,A -85,B 0,C 180,E1 24082.526,E2 24082.526} C_VEL
LIN {X 0,Y 154.039,Z 912.742,A -85,B 0,C 180,E1 24094.978,E2 24094.978} C_VEL
LIN {X 0,Y 180.437,Z 888.967,A -85,B 0,C 180,E1 24102.465,E2 24102.465} C_VEL
LIN {X 0,Y 206.958,Z 860.205,A -85,B 0,C 180,E1 24107.45,E2 24107.45} C_VEL
LIN {X 0,Y 208.069,Z 855.146,A -85,B 0,C 180,E1 24110.311,E2 24110.311} C_VEL
LIN {X 0,Y 208.164,Z 848.823,A -85,B 0,C 180,E1 24115.835,E2 24115.835} C_VEL
LIN {X 0,Y 207.789,Z 845.955,A -85,B 0,C 180,E1 24119.992,E2 24119.992} C_VEL
LIN {X 0,Y 206.221,Z 845.634,A -85,B 0,C 180,E1 24124.188,E2 24124.188} C_VEL
LIN {X 0,Y 202.856,Z 848.48,A -85,B 0,C 180,E1 24131.181,E2 24131.181} C_VEL
LIN {X 0,Y 198.752,Z 854.293,A -85,B 0,C 180,E1 24137.67,E2 24137.67} C_VEL
LIN {X 0,Y 193.485,Z 862.17,A -85,B 0,C 180,E1 24143.836,E2 24143.836} C_VEL
LIN {X 0,Y 190.48,Z 865.402,A -85,B 0,C 180,E1 24145.016,E2 24145.016} C_VEL
LIN {X 0,Y 164.99,Z 886.788,A -85,B 0,C 180,E1 24152.221,E2 24152.221} C_VEL
LIN {X 0,Y 141.973,Z 902.461,A -85,B 0,C 180,E1 24161.926,E2 24161.926} C_VEL
LIN {X 0,Y 122.131,Z 913.81,A -85,B 0,C 180,E1 24176.221,E2 24176.221} C_VEL
LIN {X 0,Y 110.476,Z 919.792,A -85,B 0,C 180,E1 24194.146,E2 24194.146} C_VEL
LIN {X 0,Y 107.833,Z 921.219,A -85,B 0,C 180,E1 24210,E2 24210} C_VEL
LIN {X 0,Y 110.502,Z 919.745,A -85,B 0,C 180,E1 24225.85,E2 24225.85} C_VEL
LIN {X 0,Y 122.164,Z 913.717,A -85,B 0,C 180,E1 24243.769,E2 24243.769} C_VEL
LIN {X 0,Y 142.046,Z 902.309,A -85,B 0,C 180,E1 24258.042,E2 24258.042} C_VEL
LIN {X 0,Y 151.389,Z 896.337,A -85,B 0,C 180,E1 24262.466,E2 24262.466} C_VEL
LIN {X 0,Y 159.505,Z 889.879,A -85,B 0,C 180,E1 24267.691,E2 24267.691} C_VEL
LIN {X 0,Y 168.356,Z 882.422,A -85,B 0,C 180,E1 24272.297,E2 24272.297} C_VEL
LIN {X 0,Y 187.755,Z 866.106,A -85,B 0,C 180,E1 24277.231,E2 24277.231} C_VEL
LIN {X 0,Y 194.05,Z 857.767,A -85,B 0,C 180,E1 24284.217,E2 24284.217} C_VEL
LIN {X 0,Y 198.472,Z 852.681,A -85,B 0,C 180,E1 24291.263,E2 24291.263} C_VEL
LIN {X 0,Y 200.646,Z 851.374,A -85,B 0,C 180,E1 24295.695,E2 24295.695} C_VEL
LIN {X 0,Y 202.47,Z 851.577,A -85,B 0,C 180,E1 24300.008,E2 24300.008} C_VEL
LIN {X 0,Y 202.588,Z 856.761,A -85,B 0,C 180,E1 24306.423,E2 24306.423} C_VEL
LIN {X 0,Y 201.925,Z 862.181,A -85,B 0,C 180,E1 24310.59,E2 24310.59} C_VEL
LIN {X 0,Y 176.34,Z 888.995,A -85,B 0,C 180,E1 24315.322,E2 24315.322} C_VEL
LIN {X 0,Y 147.707,Z 913.596,A -85,B 0,C 180,E1 24323.154,E2 24323.154} C_VEL
LIN {X 0,Y 121.136,Z 933.378,A -85,B 0,C 180,E1 24335.933,E2 24335.933} C_VEL
LIN {X 0,Y 103.238,Z 946.758,A -85,B 0,C 180,E1 24354.221,E2 24354.221} C_VEL
LIN {X 0,Y 97.658,Z 953.283,A -85,B 0,C 180,E1 24371.999,E2 24371.999} C_VEL
LIN {X 0,Y 98.532,Z 955.961,A -85,B 0,C 180,E1 24390,E2 24390} C_VEL
LIN {X 0,Y 97.673,Z 953.31,A -85,B 0,C 180,E1 24407.998,E2 24407.998} C_VEL
LIN {X 0,Y 104.86,Z 945.473,A -85,B 0,C 180,E1 24428.333,E2 24428.333} C_VEL
LIN {X 0,Y 123.449,Z 931.748,A -85,B 0,C 180,E1 24445.598,E2 24445.598} C_VEL
LIN {X 0,Y 149.208,Z 912.527,A -85,B 0,C 180,E1 24457.345,E2 24457.345} C_VEL
LIN {X 0,Y 176.562,Z 889.002,A -85,B 0,C 180,E1 24464.683,E2 24464.683} C_VEL
LIN {X 0,Y 201.129,Z 863.595,A -85,B 0,C 180,E1 24469.085,E2 24469.085} C_VEL
LIN {X 0,Y 202.237,Z 861.103,A -85,B 0,C 180,E1 24470.221,E2 24470.221} C_VEL
LIN {X 0,Y 202.723,Z 854.824,A -85,B 0,C 180,E1 24475.723,E2 24475.723} C_VEL
LIN {X 0,Y 202.48,Z 851.842,A -85,B 0,C 180,E1 24479.992,E2 24479.992} C_VEL
LIN {X 0,Y 200.744,Z 851.547,A -85,B 0,C 180,E1 24484.302,E2 24484.302} C_VEL
LIN {X 0,Y 197.287,Z 854.189,A -85,B 0,C 180,E1 24491.012,E2 24491.012} C_VEL
LIN {X 0,Y 192.562,Z 860.051,A -85,B 0,C 180,E1 24497.623,E2 24497.623} C_VEL
LIN {X 0,Y 187.978,Z 866.087,A -85,B 0,C 180,E1 24502.592,E2 24502.592} C_VEL
LIN {X 0,Y 160.965,Z 888.11,A -85,B 0,C 180,E1 24509.87,E2 24509.87} C_VEL
LIN {X 0,Y 136.874,Z 903.779,A -85,B 0,C 180,E1 24519.491,E2 24519.491} C_VEL
LIN {X 0,Y 115.695,Z 915.129,A -85,B 0,C 180,E1 24534.061,E2 24534.061} C_VEL
LIN {X 0,Y 102.993,Z 921.105,A -85,B 0,C 180,E1 24552.961,E2 24552.961} C_VEL
LIN {X 0,Y 100.043,Z 922.531,A -85,B 0,C 180,E1 24570,E2 24570} C_VEL
LIN {X 0,Y 103.021,Z 921.059,A -85,B 0,C 180,E1 24587.035,E2 24587.035} C_VEL
LIN {X 0,Y 115.731,Z 915.038,A -85,B 0,C 180,E1 24605.926,E2 24605.926} C_VEL
LIN {X 0,Y 136.954,Z 903.625,A -85,B 0,C 180,E1 24620.468,E2 24620.468} C_VEL
LIN {X 0,Y 163.942,Z 885.814,A -85,B 0,C 180,E1 24630.977,E2 24630.977} C_VEL
LIN {X 0,Y 168.356,Z 882.422,A -85,B 0,C 180,E1 24632.297,E2 24632.297} C_VEL
LIN {X 0,Y 176.16,Z 875.909,A -85,B 0,C 180,E1 24635.187,E2 24635.187} C_VEL
LIN {X 0,Y 183.509,Z 868.444,A -85,B 0,C 180,E1 24639.792,E2 24639.792} C_VEL
LIN {X 0,Y 184.805,Z 866.905,A -85,B 0,C 180,E1 24641.038,E2 24641.038} C_VEL
LIN {X 0,Y 189.415,Z 861.677,A -85,B 0,C 180,E1 24646.183,E2 24646.183} C_VEL
LIN {X 0,Y 192.523,Z 858.561,A -85,B 0,C 180,E1 24650.99,E2 24650.99} C_VEL
LIN {X 0,Y 194.963,Z 857.151,A -85,B 0,C 180,E1 24655.57,E2 24655.57} C_VEL
LIN {X 0,Y 196.907,Z 857.247,A -85,B 0,C 180,E1 24660.008,E2 24660.008} C_VEL
LIN {X 0,Y 196.793,Z 862.682,A -85,B 0,C 180,E1 24666.61,E2 24666.61} C_VEL
LIN {X 0,Y 196.376,Z 865.473,A -85,B 0,C 180,E1 24668.848,E2 24668.848} C_VEL
LIN {X 0,Y 167.307,Z 893.885,A -85,B 0,C 180,E1 24674.17,E2 24674.17} C_VEL
LIN {X 0,Y 139.192,Z 916.171,A -85,B 0,C 180,E1 24681.942,E2 24681.942} C_VEL
LIN {X 0,Y 113.878,Z 933.625,A -85,B 0,C 180,E1 24694.278,E2 24694.278} C_VEL
LIN {X 0,Y 96.641,Z 945.364,A -85,B 0,C 180,E1 24711.349,E2 24711.349} C_VEL
LIN {X 0,Y 89.968,Z 951.916,A -85,B 0,C 180,E1 24730.4,E2 24730.4} C_VEL
LIN {X 0,Y 90.662,Z 954.636,A -85,B 0,C 180,E1 24750,E2 24750} C_VEL
LIN {X 0,Y 89.982,Z 951.943,A -85,B 0,C 180,E1 24769.597,E2 24769.597} C_VEL
LIN {X 0,Y 99.71,Z 943.185,A -85,B 0,C 180,E1 24792.917,E2 24792.917} C_VEL
LIN {X 0,Y 121.495,Z 928.569,A -85,B 0,C 180,E1 24810.39,E2 24810.39} C_VEL
LIN {X 0,Y 150.134,Z 908.106,A -85,B 0,C 180,E1 24821.562,E2 24821.562} C_VEL
LIN {X 0,Y 181.026,Z 881.556,A -85,B 0,C 180,E1 24828.5,E2 24828.5} C_VEL
LIN {X 0,Y 196.489,Z 865.585,A -85,B 0,C 180,E1 24831.157,E2 24831.157} C_VEL
LIN {X 0,Y 197.019,Z 858.87,A -85,B 0,C 180,E1 24837.797,E2 24837.797} C_VEL
LIN {X 0,Y 196.229,Z 857.398,A -85,B 0,C 180,E1 24841.425,E2 24841.425} C_VEL
LIN {X 0,Y 195.069,Z 857.316,A -85,B 0,C 180,E1 24844.428,E2 24844.428} C_VEL
LIN {X 0,Y 191.089,Z 860.115,A -85,B 0,C 180,E1 24851.376,E2 24851.376} C_VEL
LIN {X 0,Y 185.964,Z 865.776,A -85,B 0,C 180,E1 24857.763,E2 24857.763} C_VEL
LIN {X 0,Y 182.819,Z 869.442,A -85,B 0,C 180,E1 24860.932,E2 24860.932} C_VEL
LIN {X 0,Y 155.738,Z 890.442,A -85,B 0,C 180,E1 24867.853,E2 24867.853} C_VEL
LIN {X 0,Y 129.464,Z 906.503,A -85,B 0,C 180,E1 24878.116,E2 24878.116} C_VEL
LIN {X 0,Y 109.45,Z 916.448,A -85,B 0,C 180,E1 24891.653,E2 24891.653} C_VEL
LIN {X 0,Y 95.567,Z 922.417,A -85,B 0,C 180,E1 24911.591,E2 24911.591} C_VEL
LIN {X 0,Y 92.259,Z 923.841,A -85,B 0,C 180,E1 24930,E2 24930} C_VEL
LIN {X 0,Y 95.95,Z 922.216,A -85,B 0,C 180,E1 24949.396,E2 24949.396} C_VEL
LIN {X 0,Y 109.486,Z 916.357,A -85,B 0,C 180,E1 24968.332,E2 24968.332} C_VEL
LIN {X 0,Y 132.112,Z 904.946,A -85,B 0,C 180,E1 24983.087,E2 24983.087} C_VEL
LIN {X 0,Y 160.302,Z 887.147,A -85,B 0,C 180,E1 24993.416,E2 24993.416} C_VEL
LIN {X 0,Y 181.542,Z 870.33,A -85,B 0,C 180,E1 24998.717,E2 24998.717} C_VEL
LIN {X 0,Y 184.805,Z 866.905,A -85,B 0,C 180,E1 25001.038,E2 25001.038} C_VEL
LIN {X 0,Y 186.345,Z 864.573,A -85,B 0,C 180,E1 25004.995,E2 25004.995} C_VEL
LIN {X 0,Y 186.956,Z 863.91,A -85,B 0,C 180,E1 25011.925,E2 25011.925} C_VEL
LIN {X 0,Y 189.046,Z 862.77,A -85,B 0,C 180,E1 25015.431,E2 25015.431} C_VEL
LIN {X 0,Y 191.226,Z 862.827,A -85,B 0,C 180,E1 25020.009,E2 25020.009} C_VEL
LIN {X 0,Y 190.716,Z 868.593,A -85,B 0,C 180,E1 25026.918,E2 25026.918} C_VEL
LIN {X 0,Y 186.811,Z 872.984,A -85,B 0,C 180,E1 25027.836,E2 25027.836} C_VEL
LIN {X 0,Y 156.921,Z 899.497,A -85,B 0,C 180,E1 25033.183,E2 25033.183} C_VEL
LIN {X 0,Y 126.385,Z 921.482,A -85,B 0,C 180,E1 25042.283,E2 25042.283} C_VEL
LIN {X 0,Y 100.72,Z 937.466,A -85,B 0,C 180,E1 25056.836,E2 25056.836} C_VEL
LIN {X 0,Y 85.124,Z 947.701,A -85,B 0,C 180,E1 25077.872,E2 25077.872} C_VEL
LIN {X 0,Y 81.612,Z 952.419,A -85,B 0,C 180,E1 25099.345,E2 25099.345} C_VEL
LIN {X 0,Y 82.78,Z 953.309,A -85,B 0,C 180,E1 25110,E2 25110} C_VEL
LIN {X 0,Y 82.367,Z 950.575,A -85,B 0,C 180,E1 25131.494,E2 25131.494} C_VEL
LIN {X 0,Y 93.814,Z 941.786,A -85,B 0,C 180,E1 25156.371,E2 25156.371} C_VEL
LIN {X 0,Y 117.614,Z 927.169,A -85,B 0,C 180,E1 25173.91,E2 25173.91} C_VEL
LIN {X 0,Y 147.368,Z 906.948,A -85,B 0,C 180,E1 25184.53,E2 25184.53} C_VEL
LIN {X 0,Y 178.408,Z 881.242,A -85,B 0,C 180,E1 25190.894,E2 25190.894} C_VEL
LIN {X 0,Y 190.788,Z 868.841,A -85,B 0,C 180,E1 25192.984,E2 25192.984} C_VEL
LIN {X 0,Y 191.223,Z 863.068,A -85,B 0,C 180,E1 25199.991,E2 25199.991} C_VEL
LIN {X 0,Y 189.141,Z 862.931,A -85,B 0,C 180,E1 25204.567,E2 25204.567} C_VEL
LIN {X 0,Y 184.822,Z 865.817,A -85,B 0,C 180,E1 25211.552,E2 25211.552} C_VEL
LIN {X 0,Y 179.304,Z 871.249,A -85,B 0,C 180,E1 25217.712,E2 25217.712} C_VEL
LIN {X 0,Y 178.167,Z 872.4,A -85,B 0,C 180,E1 25218.779,E2 25218.779} C_VEL
LIN {X 0,Y 150.713,Z 892.777,A -85,B 0,C 180,E1 25225.696,E2 25225.696} C_VEL
LIN {X 0,Y 122.154,Z 909.219,A -85,B 0,C 180,E1 25236.587,E2 25236.587} C_VEL
LIN {X 0,Y 99.576,Z 919.395,A -85,B 0,C 180,E1 25252.687,E2 25252.687} C_VEL
LIN {X 0,Y 88.196,Z 923.731,A -85,B 0,C 180,E1 25269.99,E2 25269.99} C_VEL
LIN {X 0,Y 84.469,Z 925.152,A -85,B 0,C 180,E1 25290,E2 25290} C_VEL
LIN {X 0,Y 88.217,Z 923.687,A -85,B 0,C 180,E1 25310.005,E2 25310.005} C_VEL
LIN {X 0,Y 103.452,Z 917.677,A -85,B 0,C 180,E1 25331.025,E2 25331.025} C_VEL
LIN {X 0,Y 127.581,Z 906.263,A -85,B 0,C 180,E1 25345.888,E2 25345.888} C_VEL
LIN {X 0,Y 155.407,Z 889.543,A -85,B 0,C 180,E1 25355.548,E2 25355.548} C_VEL
LIN {X 0,Y 178.134,Z 872.2,A -85,B 0,C 180,E1 25361.191,E2 25361.191} C_VEL
LIN {X 0,Y 183.828,Z 866.474,A -85,B 0,C 180,E1 25367.072,E2 25367.072} C_VEL
LIN {X 0,Y 186.956,Z 863.91,A -85,B 0,C 180,E1 25371.925,E2 25371.925} C_VEL
LIN {X 0,Y 187.309,Z 864.575,A -85,B 0,C 180,E1 25375.942,E2 25375.942} C_VEL
LIN {X 0,Y 185.292,Z 869.994,A -85,B 0,C 180,E1 25382.638,E2 25382.638} C_VEL
LIN {X 0,Y 184.986,Z 872.281,A -85,B 0,C 180,E1 25385.273,E2 25385.273} C_VEL
LIN {X 0,Y 153.499,Z 899.394,A -85,B 0,C 180,E1 25390.561,E2 25390.561} C_VEL
LIN {X 0,Y 123.468,Z 920.073,A -85,B 0,C 180,E1 25398.705,E2 25398.705} C_VEL
LIN {X 0,Y 95.956,Z 936.061,A -85,B 0,C 180,E1 25412.85,E2 25412.85} C_VEL
LIN {X 0,Y 78.279,Z 946.316,A -85,B 0,C 180,E1 25434.668,E2 25434.668} C_VEL
LIN {X 0,Y 73.741,Z 951.067,A -85,B 0,C 180,E1 25458.192,E2 25458.192} C_VEL
LIN {X 0,Y 74.872,Z 951.978,A -85,B 0,C 180,E1 25470,E2 25470} C_VEL
LIN {X 0,Y 74.86,Z 949.206,A -85,B 0,C 180,E1 25493.775,E2 25493.775} C_VEL
LIN {X 0,Y 88.28,Z 940.387,A -85,B 0,C 180,E1 25520.282,E2 25520.282} C_VEL
LIN {X 0,Y 114.205,Z 925.767,A -85,B 0,C 180,E1 25537.654,E2 25537.654} C_VEL
LIN {X 0,Y 145.61,Z 905.38,A -85,B 0,C 180,E1 25547.736,E2 25547.736} C_VEL
LIN {X 0,Y 178.05,Z 879.091,A -85,B 0,C 180,E1 25553.649,E2 25553.649} C_VEL
LIN {X 0,Y 185.077,Z 872.409,A -85,B 0,C 180,E1 25554.729,E2 25554.729} C_VEL
LIN {X 0,Y 185.391,Z 868.473,A -85,B 0,C 180,E1 25559.991,E2 25559.991} C_VEL
LIN {X 0,Y 182.124,Z 868.839,A -85,B 0,C 180,E1 25566.143,E2 25566.143} C_VEL
LIN {X 0,Y 178.23,Z 871.503,A -85,B 0,C 180,E1 25571.985,E2 25571.985} C_VEL
LIN {X 0,Y 173.386,Z 875.716,A -85,B 0,C 180,E1 25576.796,E2 25576.796} C_VEL
LIN {X 0,Y 145.75,Z 895.218,A -85,B 0,C 180,E1 25583.429,E2 25583.429} C_VEL
LIN {X 0,Y 117.649,Z 910.541,A -85,B 0,C 180,E1 25593.519,E2 25593.519} C_VEL
LIN {X 0,Y 93.476,Z 920.71,A -85,B 0,C 180,E1 25609.78,E2 25609.78} C_VEL
LIN {X 0,Y 79.911,Z 925.409,A -85,B 0,C 180,E1 25630.69,E2 25630.69} C_VEL
LIN {X 0,Y 76.685,Z 926.463,A -85,B 0,C 180,E1 25650,E2 25650} C_VEL
LIN {X 0,Y 80.933,Z 925,A -85,B 0,C 180,E1 25671.895,E2 25671.895} C_VEL
LIN {X 0,Y 97.689,Z 918.995,A -85,B 0,C 180,E1 25694.036,E2 25694.036} C_VEL
LIN {X 0,Y 123.357,Z 907.585,A -85,B 0,C 180,E1 25708.902,E2 25708.902} C_VEL
LIN {X 0,Y 152.34,Z 890.869,A -85,B 0,C 180,E1 25718.223,E2 25718.223} C_VEL
LIN {X 0,Y 172.194,Z 876.532,A -85,B 0,C 180,E1 25722.625,E2 25722.625} C_VEL
LIN {X 0,Y 178.248,Z 871.249,A -85,B 0,C 180,E1 25728.014,E2 25728.014} C_VEL
LIN {X 0,Y 182.998,Z 868.28,A -85,B 0,C 180,E1 25735.279,E2 25735.279} C_VEL
LIN {X 0,Y 185.384,Z 868.242,A -85,B 0,C 180,E1 25740.009,E2 25740.009} C_VEL
LIN {X 0,Y 185.292,Z 869.994,A -85,B 0,C 180,E1 25742.638,E2 25742.638} C_VEL
LIN {X 0,Y 182.591,Z 873.242,A -85,B 0,C 180,E1 25743.932,E2 25743.932} C_VEL
LIN {X 0,Y 168.416,Z 885.168,A -85,B 0,C 180,E1 25744.853,E2 25744.853} C_VEL
LIN {X 0,Y 136.306,Z 909.115,A -85,B 0,C 180,E1 25750.729,E2 25750.729} C_VEL
LIN {X 0,Y 102.868,Z 928.882,A -85,B 0,C 180,E1 25762.062,E2 25762.062} C_VEL
LIN {X 0,Y 78.792,Z 941.184,A -85,B 0,C 180,E1 25779.998,E2 25779.998} C_VEL
LIN {X 0,Y 67.424,Z 947.833,A -85,B 0,C 180,E1 25803.583,E2 25803.583} C_VEL
LIN {X 0,Y 66.967,Z 950.647,A -85,B 0,C 180,E1 25830,E2 25830} C_VEL
LIN {X 0,Y 67.483,Z 947.835,A -85,B 0,C 180,E1 25856.565,E2 25856.565} C_VEL
LIN {X 0,Y 83.218,Z 938.988,A -85,B 0,C 180,E1 25884.684,E2 25884.684} C_VEL
LIN {X 0,Y 111.309,Z 924.366,A -85,B 0,C 180,E1 25901.618,E2 25901.618} C_VEL
LIN {X 0,Y 143.502,Z 904.359,A -85,B 0,C 180,E1 25910.847,E2 25910.847} C_VEL
LIN {X 0,Y 175.695,Z 879.172,A -85,B 0,C 180,E1 25916.088,E2 25916.088} C_VEL
LIN {X 0,Y 179.169,Z 875.669,A -85,B 0,C 180,E1 25916.965,E2 25916.965} C_VEL
LIN {X 0,Y 179.341,Z 873.68,A -85,B 0,C 180,E1 25919.991,E2 25919.991} C_VEL
LIN {X 0,Y 176.805,Z 873.76,A -85,B 0,C 180,E1 25924.886,E2 25924.886} C_VEL
LIN {X 0,Y 171.718,Z 876.671,A -85,B 0,C 180,E1 25931.841,E2 25931.841} C_VEL
LIN {X 0,Y 168.602,Z 879.148,A -85,B 0,C 180,E1 25934.806,E2 25934.806} C_VEL
LIN {X 0,Y 138.123,Z 899.261,A -85,B 0,C 180,E1 25941.779,E2 25941.779} C_VEL
LIN {X 0,Y 110.63,Z 913.086,A -85,B 0,C 180,E1 25951.515,E2 25951.515} C_VEL
LIN {X 0,Y 87.645,Z 922.027,A -85,B 0,C 180,E1 25966.474,E2 25966.474} C_VEL
LIN {X 0,Y 73.717,Z 926.358,A -85,B 0,C 180,E1 25985.833,E2 25985.833} C_VEL
LIN {X 0,Y 68.92,Z 927.77,A -85,B 0,C 180,E1 26010,E2 26010} C_VEL
LIN {X 0,Y 73.748,Z 926.314,A -85,B 0,C 180,E1 26034.157,E2 26034.157} C_VEL
LIN {X 0,Y 92.214,Z 920.315,A -85,B 0,C 180,E1 26057.424,E2 26057.424} C_VEL
LIN {X 0,Y 119.511,Z 908.903,A -85,B 0,C 180,E1 26072.11,E2 26072.11} C_VEL
LIN {X 0,Y 149.616,Z 892.196,A -85,B 0,C 180,E1 26081.004,E2 26081.004} C_VEL
LIN {X 0,Y 168.583,Z 878.964,A -85,B 0,C 180,E1 26085.153,E2 26085.153} C_VEL
LIN {X 0,Y 173.278,Z 875.346,A -85,B 0,C 180,E1 26089.98,E2 26089.98} C_VEL
LIN {X 0,Y 176.73,Z 873.596,A -85,B 0,C 180,E1 26095.112,E2 26095.112} C_VEL
LIN {X 0,Y 179.336,Z 873.461,A -85,B 0,C 180,E1 26100.009,E2 26100.009} C_VEL
LIN {X 0,Y 179.117,Z 875.5,A -85,B 0,C 180,E1 26103.037,E2 26103.037} C_VEL
LIN {X 0,Y 173.978,Z 880.435,A -85,B 0,C 180,E1 26104.094,E2 26104.094} C_VEL
LIN {X 0,Y 168.416,Z 885.168,A -85,B 0,C 180,E1 26104.853,E2 26104.853} C_VEL
LIN {X 0,Y 154.229,Z 895.429,A -85,B 0,C 180,E1 26105.466,E2 26105.466} C_VEL
LIN {X 0,Y 141.297,Z 903.576,A -85,B 0,C 180,E1 26106.09,E2 26106.09} C_VEL
LIN {X 0,Y 139.57,Z 904.69,A -85,B 0,C 180,E1 26106.386,E2 26106.386} C_VEL
LIN {X 0,Y 106.57,Z 924.13,A -85,B 0,C 180,E1 26115.071,E2 26115.071} C_VEL
LIN {X 0,Y 76.123,Z 938.738,A -85,B 0,C 180,E1 26132.697,E2 26132.697} C_VEL
LIN {X 0,Y 60.258,Z 946.426,A -85,B 0,C 180,E1 26159.944,E2 26159.944} C_VEL
LIN {X 0,Y 59.053,Z 949.315,A -85,B 0,C 180,E1 26190,E2 26190} C_VEL
LIN {X 0,Y 60.28,Z 946.458,A -85,B 0,C 180,E1 26220.044,E2 26220.044} C_VEL
LIN {X 0,Y 78.581,Z 937.638,A -85,B 0,C 180,E1 26249.544,E2 26249.544} C_VEL
LIN {X 0,Y 108.981,Z 922.969,A -85,B 0,C 180,E1 26265.753,E2 26265.753} C_VEL
LIN {X 0,Y 142.432,Z 902.93,A -85,B 0,C 180,E1 26274.171,E2 26274.171} C_VEL
LIN {X 0,Y 173.1,Z 879.513,A -85,B 0,C 180,E1 26278.745,E2 26278.745} C_VEL
LIN {X 0,Y 173.194,Z 878.763,A -85,B 0,C 180,E1 26279.99,E2 26279.99} C_VEL
LIN {X 0,Y 170.257,Z 878.956,A -85,B 0,C 180,E1 26285.075,E2 26285.075} C_VEL
LIN {X 0,Y 164.885,Z 881.867,A -85,B 0,C 180,E1 26291.827,E2 26291.827} C_VEL
LIN {X 0,Y 163.587,Z 882.75,A -85,B 0,C 180,E1 26292.946,E2 26292.946} C_VEL
LIN {X 0,Y 132.094,Z 902.396,A -85,B 0,C 180,E1 26299.533,E2 26299.533} C_VEL
LIN {X 0,Y 103.755,Z 915.62,A -85,B 0,C 180,E1 26309.234,E2 26309.234} C_VEL
LIN {X 0,Y 77.532,Z 924.723,A -85,B 0,C 180,E1 26327.063,E2 26327.063} C_VEL
LIN {X 0,Y 62.648,Z 928.697,A -85,B 0,C 180,E1 26356.062,E2 26356.062} C_VEL
LIN {X 0,Y 63.8,Z 928.37,A -85,B 0,C 180,E1 26388.992,E2 26388.992} C_VEL
LIN {X 0,Y 82.159,Z 923.277,A -85,B 0,C 180,E1 26417.279,E2 26417.279} C_VEL
LIN {X 0,Y 109.839,Z 913.045,A -85,B 0,C 180,E1 26433.25,E2 26433.25} C_VEL
LIN {X 0,Y 142.178,Z 896.558,A -85,B 0,C 180,E1 26442.786,E2 26442.786} C_VEL
LIN {X 0,Y 163.617,Z 882.527,A -85,B 0,C 180,E1 26447.026,E2 26447.026} C_VEL
LIN {X 0,Y 167.822,Z 879.859,A -85,B 0,C 180,E1 26451.525,E2 26451.525} C_VEL
LIN {X 0,Y 170.446,Z 878.762,A -85,B 0,C 180,E1 26455.433,E2 26455.433} C_VEL
LIN {X 0,Y 173.112,Z 879.069,A -85,B 0,C 180,E1 26460.828,E2 26460.828} C_VEL
LIN {X 0,Y 173.077,Z 879.325,A -85,B 0,C 180,E1 26461.237,E2 26461.237} C_VEL
LIN {X 0,Y 140.664,Z 903.963,A -85,B 0,C 180,E1 26466.17,E2 26466.17} C_VEL
LIN {X 0,Y 139.57,Z 904.69,A -85,B 0,C 180,E1 26466.386,E2 26466.386} C_VEL
LIN {X 0,Y 132.304,Z 909.105,A -85,B 0,C 180,E1 26467.296,E2 26467.296} C_VEL
LIN {X 0,Y 110.819,Z 919.691,A -85,B 0,C 180,E1 26468.944,E2 26468.944} C_VEL
LIN {X 0,Y 109.01,Z 920.566,A -85,B 0,C 180,E1 26469.392,E2 26469.392} C_VEL
LIN {X 0,Y 77.661,Z 934.986,A -85,B 0,C 180,E1 26482.889,E2 26482.889} C_VEL
LIN {X 0,Y 56.13,Z 943.769,A -85,B 0,C 180,E1 26507.771,E2 26507.771} C_VEL
LIN {X 0,Y 50.312,Z 946.995,A -85,B 0,C 180,E1 26532.547,E2 26532.547} C_VEL
LIN {X 0,Y 51.12,Z 947.979,A -85,B 0,C 180,E1 26550,E2 26550} C_VEL
LIN {X 0,Y 53.339,Z 945.078,A -85,B 0,C 180,E1 26584.458,E2 26584.458} C_VEL
LIN {X 0,Y 73.31,Z 936.812,A -85,B 0,C 180,E1 26614.01,E2 26614.01} C_VEL
LIN {X 0,Y 104.898,Z 922.738,A -85,B 0,C 180,E1 26629.371,E2 26629.371} C_VEL
LIN {X 0,Y 139.988,Z 902.702,A -85,B 0,C 180,E1 26637.231,E2 26637.231} C_VEL
LIN {X 0,Y 165.997,Z 884.04,A -85,B 0,C 180,E1 26640.558,E2 26640.558} C_VEL
LIN {X 0,Y 163.58,Z 884.013,A -85,B 0,C 180,E1 26645.282,E2 26645.282} C_VEL
LIN {X 0,Y 159.902,Z 885.649,A -85,B 0,C 180,E1 26649.891,E2 26649.891} C_VEL
LIN {X 0,Y 156.111,Z 888.18,A -85,B 0,C 180,E1 26651.214,E2 26651.214} C_VEL
LIN {X 0,Y 122.847,Z 907.141,A -85,B 0,C 180,E1 26657.961,E2 26657.961} C_VEL
LIN {X 0,Y 93.406,Z 919.417,A -85,B 0,C 180,E1 26668.303,E2 26668.303} C_VEL
LIN {X 0,Y 67.379,Z 927.215,A -85,B 0,C 180,E1 26687.789,E2 26687.789} C_VEL
LIN {X 0,Y 55.113,Z 930.009,A -85,B 0,C 180,E1 26714.11,E2 26714.11} C_VEL
LIN {X 0,Y 55.126,Z 929.985,A -85,B 0,C 180,E1 26745.887,E2 26745.887} C_VEL
LIN {X 0,Y 72.023,Z 925.969,A -85,B 0,C 180,E1 26777.164,E2 26777.164} C_VEL
LIN {X 0,Y 100.212,Z 916.816,A -85,B 0,C 180,E1 26794.62,E2 26794.62} C_VEL
LIN {X 0,Y 133.165,Z 901.722,A -85,B 0,C 180,E1 26804.407,E2 26804.407} C_VEL
LIN {X 0,Y 157.562,Z 887.011,A -85,B 0,C 180,E1 26808.969,E2 26808.969} C_VEL
LIN {X 0,Y 160.862,Z 884.928,A -85,B 0,C 180,E1 26811.156,E2 26811.156} C_VEL
LIN {X 0,Y 164.94,Z 883.597,A -85,B 0,C 180,E1 26816.949,E2 26816.949} C_VEL
LIN {X 0,Y 165.998,Z 883.82,A -85,B 0,C 180,E1 26819.399,E2 26819.399} C_VEL
LIN {X 0,Y 130.535,Z 908.513,A -85,B 0,C 180,E1 26824.401,E2 26824.401} C_VEL
LIN {X 0,Y 109.01,Z 920.566,A -85,B 0,C 180,E1 26829.392,E2 26829.392} C_VEL
LIN {X 0,Y 93.307,Z 927.047,A -85,B 0,C 180,E1 26831.889,E2 26831.889} C_VEL
LIN {X 0,Y 77.569,Z 932.553,A -85,B 0,C 180,E1 26835.552,E2 26835.552} C_VEL
LIN {X 0,Y 50.348,Z 942.385,A -85,B 0,C 180,E1 26861.472,E2 26861.472} C_VEL
LIN {X 0,Y 42.676,Z 945.635,A -85,B 0,C 180,E1 26889.293,E2 26889.293} C_VEL
LIN {X 0,Y 43.179,Z 946.642,A -85,B 0,C 180,E1 26910,E2 26910} C_VEL
LIN {X 0,Y 46.808,Z 943.698,A -85,B 0,C 180,E1 26950.147,E2 26950.147} C_VEL
LIN {X 0,Y 73.997,Z 933.942,A -85,B 0,C 180,E1 26982.542,E2 26982.542} C_VEL
LIN {X 0,Y 110.747,Z 917.918,A -85,B 0,C 180,E1 26995.611,E2 26995.611} C_VEL
LIN {X 0,Y 147.176,Z 896.507,A -85,B 0,C 180,E1 27001.49,E2 27001.49} C_VEL
LIN {X 0,Y 158.452,Z 888.427,A -85,B 0,C 180,E1 27003.003,E2 27003.003} C_VEL
LIN {X 0,Y 154.926,Z 889.535,A -85,B 0,C 180,E1 27007.802,E2 27007.802} C_VEL
LIN {X 0,Y 150.843,Z 891.972,A -85,B 0,C 180,E1 27008.935,E2 27008.935} C_VEL
LIN {X 0,Y 118.057,Z 909.67,A -85,B 0,C 180,E1 27015.035,E2 27015.035} C_VEL
LIN {X 0,Y 84.307,Z 922.594,A -85,B 0,C 180,E1 27026.499,E2 27026.499} C_VEL
LIN {X 0,Y 61.805,Z 928.531,A -85,B 0,C 180,E1 27042.907,E2 27042.907} C_VEL
LIN {X 0,Y 47.557,Z 931.346,A -85,B 0,C 180,E1 27072.032,E2 27072.032} C_VEL
LIN {X 0,Y 47.688,Z 931.296,A -85,B 0,C 180,E1 27108.447,E2 27108.447} C_VEL
LIN {X 0,Y 66.951,Z 927.287,A -85,B 0,C 180,E1 27142.079,E2 27142.079} C_VEL
LIN {X 0,Y 97.113,Z 918.138,A -85,B 0,C 180,E1 27158.798,E2 27158.798} C_VEL
LIN {X 0,Y 131.283,Z 903.047,A -85,B 0,C 180,E1 27167.69,E2 27167.69} C_VEL
LIN {X 0,Y 152.663,Z 890.653,A -85,B 0,C 180,E1 27171.281,E2 27171.281} C_VEL
LIN {X 0,Y 156.64,Z 888.71,A -85,B 0,C 180,E1 27174.483,E2 27174.483} C_VEL
LIN {X 0,Y 158.437,Z 888.247,A -85,B 0,C 180,E1 27176.987,E2 27176.987} C_VEL
LIN {X 0,Y 126.185,Z 909.394,A -85,B 0,C 180,E1 27181.379,E2 27181.379} C_VEL
LIN {X 0,Y 91.819,Z 926.643,A -85,B 0,C 180,E1 27189.575,E2 27189.575} C_VEL
LIN {X 0,Y 77.569,Z 932.553,A -85,B 0,C 180,E1 27195.552,E2 27195.552} C_VEL
LIN {X 0,Y 62.026,Z 936.969,A -85,B 0,C 180,E1 27201.237,E2 27201.237} C_VEL
LIN {X 0,Y 47.288,Z 940.359,A -85,B 0,C 180,E1 27210.661,E2 27210.661} C_VEL
LIN {X 0,Y 35.203,Z 944.269,A -85,B 0,C 180,E1 27244.618,E2 27244.618} C_VEL
LIN {X 0,Y 35.217,Z 945.302,A -85,B 0,C 180,E1 27270,E2 27270} C_VEL
LIN {X 0,Y 40.865,Z 942.314,A -85,B 0,C 180,E1 27317.605,E2 27317.605} C_VEL
LIN {X 0,Y 71.697,Z 932.627,A -85,B 0,C 180,E1 27348.757,E2 27348.757} C_VEL
LIN {X 0,Y 108.1,Z 917.605,A -85,B 0,C 180,E1 27359.501,E2 27359.501} C_VEL
LIN {X 0,Y 145.178,Z 896.748,A -85,B 0,C 180,E1 27364.476,E2 27364.476} C_VEL
LIN {X 0,Y 150.046,Z 893.382,A -85,B 0,C 180,E1 27365.201,E2 27365.201} C_VEL
LIN {X 0,Y 148.015,Z 894.421,A -85,B 0,C 180,E1 27366.206,E2 27366.206} C_VEL
LIN {X 0,Y 112.338,Z 912.759,A -85,B 0,C 180,E1 27372.148,E2 27372.148} C_VEL
LIN {X 0,Y 79.209,Z 924.46,A -85,B 0,C 180,E1 27382.372,E2 27382.372} C_VEL
LIN {X 0,Y 56.77,Z 929.846,A -85,B 0,C 180,E1 27397.116,E2 27397.116} C_VEL
LIN {X 0,Y 40.348,Z 932.633,A -85,B 0,C 180,E1 27428.038,E2 27428.038} C_VEL
LIN {X 0,Y 40.374,Z 932.607,A -85,B 0,C 180,E1 27471.947,E2 27471.947} C_VEL
LIN {X 0,Y 62.443,Z 928.607,A -85,B 0,C 180,E1 27507.758,E2 27507.758} C_VEL
LIN {X 0,Y 94.565,Z 919.459,A -85,B 0,C 180,E1 27523.222,E2 27523.222} C_VEL
LIN {X 0,Y 126.239,Z 906.185,A -85,B 0,C 180,E1 27530.456,E2 27530.456} C_VEL
LIN {X 0,Y 147.237,Z 894.71,A -85,B 0,C 180,E1 27533.614,E2 27533.614} C_VEL
LIN {X 0,Y 149.661,Z 893.473,A -85,B 0,C 180,E1 27534.838,E2 27534.838} C_VEL
LIN {X 0,Y 115.18,Z 913.925,A -85,B 0,C 180,E1 27539.226,E2 27539.226} C_VEL
LIN {X 0,Y 79.879,Z 929.58,A -85,B 0,C 180,E1 27547.868,E2 27547.868} C_VEL
LIN {X 0,Y 47.288,Z 940.359,A -85,B 0,C 180,E1 27570.661,E2 27570.661} C_VEL
LIN {X 0,Y 37.748,Z 942.264,A -85,B 0,C 180,E1 27582.656,E2 27582.656} C_VEL
LIN {X 0,Y 26.517,Z 943.563,A -85,B 0,C 180,E1 27617.697,E2 27617.697} C_VEL
LIN {X 0,Y 27.227,Z 943.957,A -85,B 0,C 180,E1 27630,E2 27630} C_VEL
LIN {X 0,Y 35.845,Z 940.931,A -85,B 0,C 180,E1 27687.346,E2 27687.346} C_VEL
LIN {X 0,Y 67.307,Z 932.278,A -85,B 0,C 180,E1 27714.202,E2 27714.202} C_VEL
LIN {X 0,Y 105.833,Z 917.346,A -85,B 0,C 180,E1 27723.552,E2 27723.552} C_VEL
LIN {X 0,Y 121.292,Z 909.773,A -85,B 0,C 180,E1 27725.57,E2 27725.57} C_VEL
